(* CODESYS project lclspmps.library
   Company: SLAC
   Version: 0.0.0
   Placeholder: LCLS PMPS
   Title: LCLS PMPS

Project tree, tasks and I/O mapping:
  libraries: LCLS General, * (SLAC); Tc2_MC2, * (Beckhoff Automation GmbH); Tc2_Standard, * (Beckhoff Automation GmbH); Tc2_System, * (Beckhoff Automation GmbH); Tc2_Utilities, * (Beckhoff Automation GmbH); Tc3_Module, * (Beckhoff Automation GmbH); TcUnit, * (www.tcunit.org); VisuDialogs, * (System); VisuSymbols, 3.5.10.0 (System)
  DUTs/
    data type E_ExampleDeviceStates
    data type ST_BeamParams
    data type ST_BinarySolidAttenuator
    data type ST_Device
    data type ST_DeviceState
    data type ST_DeviceStateExt
    data type ST_SolidAttenuatorBlade
  GVLs/
    global variables GVL
    global variables PMPS_GVL_BeamParams
  POUs/
    DeviceImplementationEx1/
      function block FB_ExampleDevice [FBD]: Initialize
      function block FB_ExampleDeviceSM [UML]: AwaitingBeamParameters_ENTRY, ExecutingMove_DO, Moving_ENTRY, Moving_EXIT, NewMove_ENTRY, Stopping_ENTRY, Stopping_EXIT
    DeviceImplementationEx2/
      function block FB_ExampleDeviceSM_All [UML]: Always_DO, AwaitingBeamParameters_ENTRY, Init, MoveComplete_ENTRY, Moving_ENTRY, Moving_EXIT, NewMove_ENTRY, Stopping_ENTRY, Stopping_EXIT, VerifyingNewTargetState_DO
    FlatMirrorEx/
    HelperFunctions/
      function F_DeviceState_To_DeviceStateExt [ST]
      function F_DifferentBeamParams [ST]
      function F_eVWithinSpec [ST]
      function F_SafeBPCompare [ST]
      function F_SetBeamParams [ST]
      function F_SetStateParams [ST]
    MajorComponents/
      function block BeamParameterTransitionManager [UML]: AcquiringSafeBeamParams_DO, AssertFinalBP, AssertTransitionBP, AuthorizeTransition, DeauthorizeMove, DeauthorizeTransition, RemoveTransitionAssertion, RemoveTransitionAuthorization, SetNewTarget, WaitingForFinalAssertion_DO, WaitingForFinalAssertion_EXIT, WaitingForTransitionAssertion_DO, WaitingForTransitionAssertion_EXIT
      function block FB_Arbiter [ST]: A_Init, AddRequest, ArbitrateBP, CheckRequest, GetArbitratedBP, RemoveRequest
      function block FB_BeamClassOutputs [ST]
      function block FB_BeamParamAssertionPool [ST]: A_Add, A_Count, A_GetFirst, A_GetNext, A_Lookup, A_Remove, A_Reset
      function block FB_FastFault [ST]
      function block FB_HardwareFFOutput [ST]: CheckIn, EvaluateOutput, Register
      function block FB_LinearDeviceStateTable [ST]: A_Add, A_Count, A_GetFirst, A_GetNext, A_Lookup, A_Remove, A_Reset
      function block FB_LinearGovernor [ST]
      function block FB_PhotonEnergyWatcher [ST]
      function block FB_UsualSuspects [ST]: M_Register
    TestComponents/
      function block FB_Arbiter_Test [ST]: Arbitration, FB_init, RequestCheckRemoveBP, RunTests
      function block FB_AttenuatorSimulator [ST]
      function block FB_BPTM_Test [ST]: BPTMBasicFunction, FB_init, RunTests
      function block FB_eVWithinSpec_Test [ST]: evWithinRangeChecks, FB_init, RunTests
      function block FB_FastFault_Test [ST]: FB_init, FFCombinedFunctionality, FFRegistration, RunTests
      function block FB_MachineSimulator [ST]
      function block FB_PhotonEnergyWatcher_Test [ST]: FB_init, PEWatcherBasicFunction, RunTests
      function block FB_SafeBPCompare_Test [ST]: BeamOffIsSafe, BPComparisonCheck, FB_init, RunTests
      function block FB_SolidAttenuator [ST]
    program Fast_Faults [ST]
    program Fast_Faults_Evaluate [ST]
    program MachineSimulation [ST]
    program MAIN [ST]: Initialize
    program PMPS_Arbiter [ST]
    program TestSetups [ST]
  VISUs/
    visualisation ArbiterStats
    visualisation FastFaultGUI
    visualisation ImagerGUI
    visualisation PhotonEnergyWatcher
    visualisation Visualization
  text list GlobalTextList
  image pool ImagePool
  00000000-0000-0000-0000-000000000000|MPS Architecture.png
*)

// DUTs/E_ExampleDeviceStates
{attribute 'qualified_only'}
{attribute 'strict'}
TYPE E_ExampleDeviceStates :
(
	enum_member := 0
);
END_TYPE

// DUTs/ST_BeamParams
TYPE ST_BeamParams :
STRUCT
	// Beam parameters
	// These must be filled in by the caller.
	
	//Note: fAtt is a local parameter, meaning it is distributed to the nearest
	// upstream attenuator component.
	fAtt : REAL := 100; //Requested attenuation %
	
	
	
	//Machine parameters
	nBeamClass	:	BYTE := 16#F;
	nRate	:	UDINT	:= 10; //Pulse-rate
	fPP_mJ : REAL := 20; //Per pulse max energy (mJ)
	//1.5-0keV subdivided per bit
	(*
	0.0-0.2 - 0 (lsb)
	0.2-0.3 - 1
	0.3-0.4 - 2
	0.4-0.5 - 3
	0.5-0.6 - 4
	0.6-0.7 - 5
	0.7-0.8 - 6
	0.8-0.9 - 7
	0.9-1.0 - 8
	1.0-1.1 - 9
	1.1-1.2 - 10
	1.2-1.3 - 11
	1.3-1.4 - 12
	1.4-1.5 - 13 (msb)
	na - 14
	na - 15
	*)
	
	{attribute 'displaymode':='binary'}
	neVReqRange	:	WORD	:= 2#1111_1111_1111_1111; //Valid photon energy ranges
	
	reV	:	REAL	:=0; //Photon energy (calculated by undulator gap)

END_STRUCT
END_TYPE

// DUTs/ST_BinarySolidAttenuator
TYPE ST_BinarySolidAttenuator :
STRUCT
	axBlades	: ARRAY [0..9] OF ST_SolidAttenuatorBlade;
END_STRUCT
END_TYPE

// DUTs/ST_Device
TYPE ST_Device :
STRUCT
	//IO
	stAxis	:	AXIS_REF;
	//The following limit switches must be TRUE or high (ie. NC) to enable that direction of motion
	//The EPICS display should show an inverted indicator to communicate end of travel reached
	i_xLoLim	AT %I*	:	BOOL; //Wire normally-closed
	i_xHiLim	AT %I*	:	BOOL; //Wire normally-closed
	
	//Acuator Parameters
	lrUpperPositionLimit	:	LREAL := 10000000000; //Use in conjuntion with limit switches or set to a huge number to ignore
	lrLowerPositionLimit	:	LREAL := -10000000000; //Use in conjuntion with limit switches or set to a huge number to ignore
	
	xEnable	:	BOOL := TRUE;
	
	//Supervisory System
	
	//MPS Override
	xOverrideMPSLimits	: BOOL := FALSE; //Set true to move beyond MPS limits. Note this will trip beam off.
	
	//Status and Faults
	xClearFaults	:	BOOL;	//Rising edge tries to clear faults of all kinds
	
	xGovernorFault	:	BOOL;	//Indicates governor is faulted
	xGovernorOverridden	:	BOOL; //Indicates governor is in override mode
	xSMFault		:	BOOL;	//Indicates component state machine is faulted
	
	//Device States
	StateTable		:	FB_LinearDeviceStateTable;
	
	stTransitionState	:	ST_DeviceState; //The transition state might have non-zero beam parameters
	nSafeState			:	UDINT; //State where the device is considered safe
	nTransitionState	:	UDINT;
	
	nRequestedState	:	UDINT; //EPICS control, cleaned (checked against array limits) and deposited in nTargetState
	nTargetState	:	UDINT; //The requested state should be deposited here after cleaning
	nActiveState	:	UDINT; //The last successfully reached state
	
	
END_STRUCT
END_TYPE

// DUTs/ST_DeviceState
TYPE ST_DeviceState :
STRUCT
	
	//State name
	sStateName	:	STRING;
	nStateRef	:	UDINT; //Primary key of device state database
	
	//////////////////
	// This stuff may belong in a sub-class or something
	//Position
	rPosition	:	REAL := 0; //Center of the state
	//Tolerance
	rTolerance :	REAL := 0; //+/- amount
	//////////////////
	//Required beam parameters
	stReqBeamParam	:	ST_BeamParams;

END_STRUCT
END_TYPE

// DUTs/ST_DeviceStateExt
//Use when working with states in code
//Extended with a valid boolean to indicate the structure was loaded
//properly
TYPE ST_DeviceStateExt EXTENDS ST_DeviceState :
STRUCT
	xValid	:	BOOL := FALSE;
END_STRUCT
END_TYPE

// DUTs/ST_SolidAttenuatorBlade
TYPE ST_SolidAttenuatorBlade :
STRUCT
	xRequestedIn	:	BOOL;
	xCurrentIn	:	BOOL;
	rThickness	:	REAL;
END_STRUCT
END_TYPE

// GVLs/GVL

VAR_GLOBAL
	g_fbArbiter	:	FB_Arbiter;
	g_FastFaultOutput1	:	FB_HardwareFFOutput;
	g_rTestingVelocity	:	LREAL := VISIBLE_TEST_VELOCITY;
	g_fbFFRegistry	:	FB_UsualSuspects;
END_VAR

VAR_GLOBAL CONSTANT
	EXCLUDED_ASSERTION_ID	:	UDINT	:= 16#FFFFFFFF; //An assertion ID that should always return "not found" in the assertion pool
	VISIBLE_TEST_VELOCITY	:	LREAL	:= 10;
	FAST_TEST_VELOCITY		:	LREAL	:= 100;
	MAX_DEVICE_STATES		:	UDINT	:= 300;
END_VAR

// GVLs/PMPS_GVL_BeamParams
{attribute 'qualified_only'}
VAR_GLOBAL
	stReqFBDBeamParamsSum	:	ST_BeamParams;
	stReqMethBeamParamSum	:	ST_BeamParams;
	stCurrentBeamParameters	:	ST_BeamParams;
END_VAR
VAR_GLOBAL CONSTANT
	cstFullBeam	:	ST_BeamParams := (
		fAtt := 0,
		fPP_mJ := 1E4,
		neVReqRange := 2#1111_1111_1111_1111,
		nRate	:= UDINT#1000000
		
);
	cstSafeBeam	:	ST_BeamParams := (
		fAtt := 100,
		fPP_mJ := 0,
		neVReqRange := 0,
		nRate	:= 0
);
	cnMaxStateArrayLen : INT := 20;
	
	MAX_ASSERIONS	:	UDINT := 100; //Maximum number of assertions permitted in the arbiter
	
	g_cBoundaries	:	INT	:= 15;
	g_areVBoundaries	:	ARRAY [0..g_cBoundaries]	OF	REAL	:= [
	0.2,
	0.3,
	0.4,
	0.5,
	0.6,
	0.7,
	0.8,
	0.9,
	1.0,
	1.1,
	1.2,
	1.3,
	1.4,
	1.5,
	1.6
];
END_VAR

// POUs/DeviceImplementationEx1/FB_ExampleDevice
FUNCTION_BLOCK FB_ExampleDevice
VAR_INPUT
END_VAR
VAR_OUTPUT
END_VAR
VAR
	MC_MoveAbsolute_0: MC_MoveAbsolute;
	fbBCTM: BeamParameterTransitionManager;
	FB_ExampleDeviceSM_0: FB_ExampleDeviceSM;
	stDevice	:	ST_Device;
	MC_Power_0: MC_Power;
	MC_Stop_0	:	MC_Stop;
END_VAR

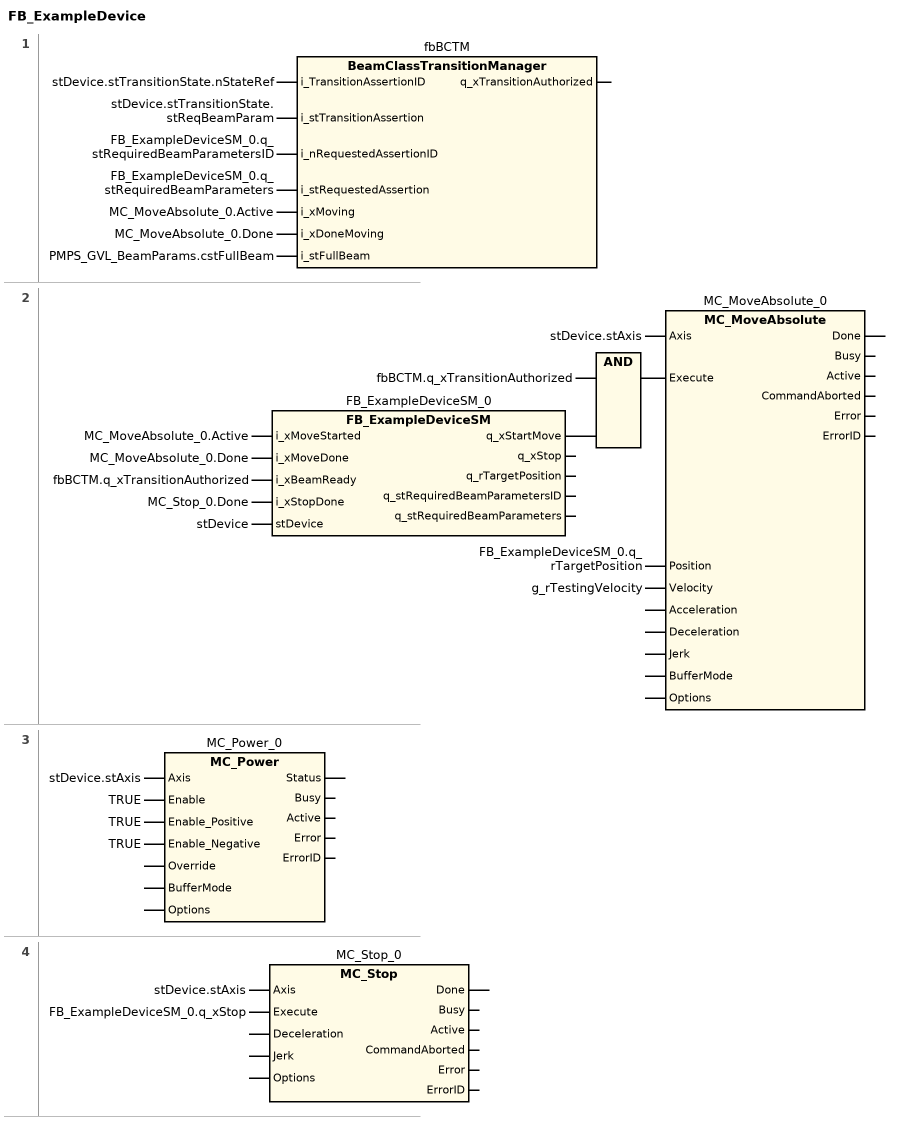
// NETWORK 1
fbBCTM(
    i_TransitionAssertionID := stDevice.stTransitionState.nStateRef,
    i_stTransitionAssertion := stDevice.stTransitionState.stReqBeamParam,
    i_nRequestedAssertionID := FB_ExampleDeviceSM_0.q_stRequiredBeamParametersID,
    i_stRequestedAssertion := FB_ExampleDeviceSM_0.q_stRequiredBeamParameters,
    i_xMoving := MC_MoveAbsolute_0.Active,
    i_xDoneMoving := MC_MoveAbsolute_0.Done,
    i_stFullBeam := PMPS_GVL_BeamParams.cstFullBeam); // BeamClassTransitionManager

// NETWORK 2
FB_ExampleDeviceSM_0(
    i_xMoveStarted := MC_MoveAbsolute_0.Active,
    i_xMoveDone := MC_MoveAbsolute_0.Done,
    i_xBeamReady := fbBCTM.q_xTransitionAuthorized,
    i_xStopDone := MC_Stop_0.Done,
    stDevice := stDevice); // FB_ExampleDeviceSM
MC_MoveAbsolute_0(
    Axis := stDevice.stAxis,
    Execute := fbBCTM.q_xTransitionAuthorized AND FB_ExampleDeviceSM_0.q_xStartMove,
    Position := FB_ExampleDeviceSM_0.q_rTargetPosition,
    Velocity := g_rTestingVelocity); // MC_MoveAbsolute

// NETWORK 3
MC_Power_0(Axis := stDevice.stAxis, Enable := TRUE, Enable_Positive := TRUE, Enable_Negative := TRUE); // MC_Power

// NETWORK 4
MC_Stop_0(Axis := stDevice.stAxis, Execute := FB_ExampleDeviceSM_0.q_xStop); // MC_Stop

ACTION Initialize:

stDevice.astStates[1].rPosition := 100;
stDevice.astStates[1].nStateRef := 16#1;
stDevice.astStates[1].stReqBeamParam := F_SetBeamParams(
	fAtt := 20,
	fPP_mJ := 1,
	fLower_eV := 0,
	fUpper_eV := 1500
);

stDevice.astStates[2].rPosition := 200;
stDevice.astStates[2].nStateRef := 16#2;
stDevice.astStates[2].stReqBeamParam := F_SetBeamParams(
	fAtt := 50,
	fPP_mJ := 1,
	fLower_eV := 0,
	fUpper_eV := 1500
);

stDevice.astStates[3].rPosition := 300;
stDevice.astStates[3].nStateRef := 16#3;
stDevice.astStates[3].stReqBeamParam := F_SetBeamParams(
	fAtt := 50,
	fPP_mJ := 0.5,
	fLower_eV := 0,
	fUpper_eV := 1500
);

stDevice.stTransitionState.nStateRef := 16#10;
stDevice.stTransitionState.stReqBeamParam := F_SetBeamParams(
	fAtt := 100,
	fPP_mJ := 1,
	fLower_eV := 0,
	fUpper_eV := 1500
);
END_ACTION

END_FUNCTION_BLOCK

// POUs/DeviceImplementationEx1/FB_ExampleDeviceSM

FUNCTION_BLOCK FB_ExampleDeviceSM
VAR_INPUT
	i_xMoveStarted	:	BOOL; //Connect to moving flag
	i_xMoveDone	:	BOOL; //Connect to move done flag
	i_xBeamReady	:	BOOL; //Connect to transitioneer
	i_xStopDone	:	BOOL; //Connect to MC_Stop.Done
END_VAR
VAR_OUTPUT
	q_xStartMove	:	BOOL; //Connect to MC_Absolute.Execute
	q_xStop			:	BOOL; //Connect to MC_Stop.Execute
	q_rTargetPosition	:	REAL; //Connect to MC_Absolute.Position
	q_stRequiredBeamParametersID	:	UDINT;
	q_stRequiredBeamParameters	:	ST_BeamParams; //Connect to BeamParameterTransitionManager
END_VAR
VAR_IN_OUT
	stDevice	:	ST_Device;
END_VAR
VAR
	nTargetState	:	INT;
	
	xNewReq	:	BOOL; //Set true when new target request present
	
END_VAR

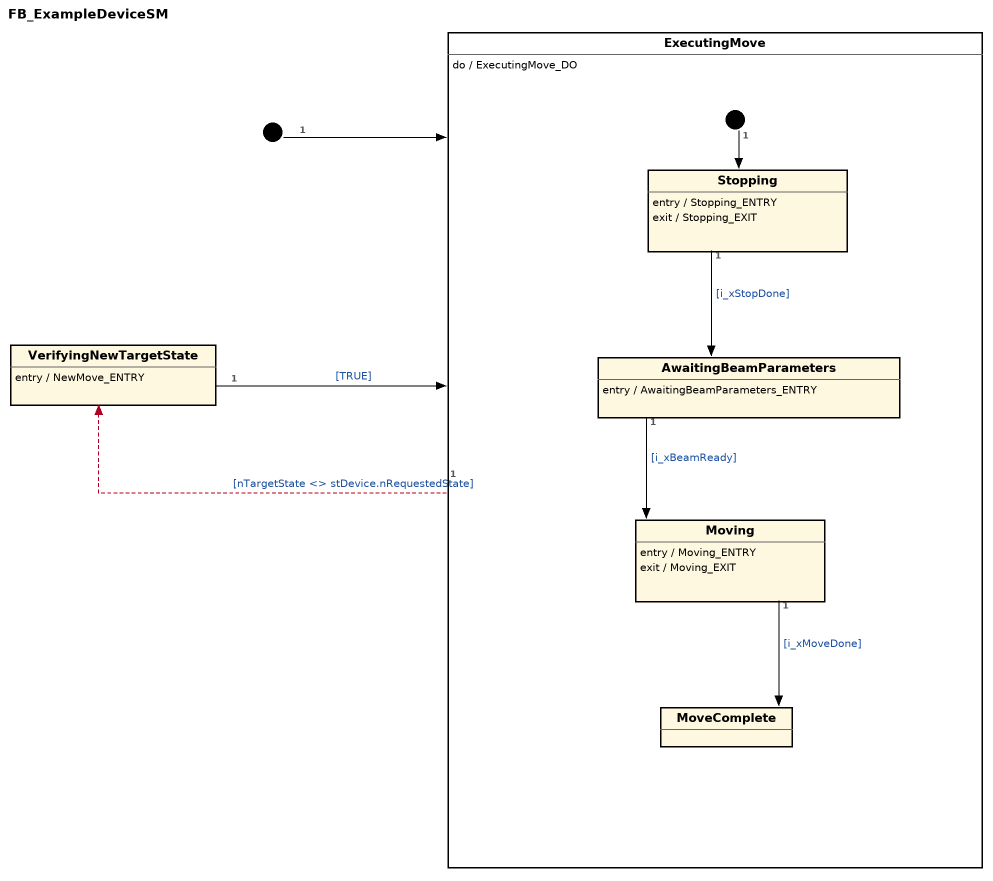
STATECHART FB_ExampleDeviceSM  // abortable
    START StartState1
    COMPOSITE STATE ExecutingMove
        do / ExecutingMove_DO
        START StartState2
        STATE Stopping
            entry / Stopping_ENTRY
            exit / Stopping_EXIT
        STATE AwaitingBeamParameters
            entry / AwaitingBeamParameters_ENTRY
        STATE Moving
            entry / Moving_ENTRY
            exit / Moving_EXIT
        STATE MoveComplete
        StartState2 -> Stopping  // priority 1, on completion
        Stopping -> AwaitingBeamParameters [i_xStopDone] // priority 1, rising edge
        AwaitingBeamParameters -> Moving [i_xBeamReady] // priority 1, rising edge
        Moving -> MoveComplete [i_xMoveDone] // priority 1, rising edge
    END_STATE
    STATE VerifyingNewTargetState
        entry / NewMove_ENTRY
    StartState1 -> ExecutingMove  // priority 1, on completion
    ExecutingMove -> VerifyingNewTargetState [nTargetState <> stDevice.nRequestedState] // priority 1, exception, rising edge
    VerifyingNewTargetState -> ExecutingMove [TRUE] // priority 1
END_STATECHART

ACTION AwaitingBeamParameters_ENTRY:
q_stRequiredBeamParameters := stDevice.astStates[nTargetState].stReqBeamParam;
q_stRequiredBeamParametersID := stDevice.astStates[nTargetState].nStateRef;
END_ACTION

ACTION ExecutingMove_DO:

END_ACTION

ACTION Moving_ENTRY:
q_xStartMove := TRUE;
q_rTargetPosition := stDevice.astStates[nTargetState].rPosition;
END_ACTION

ACTION Moving_EXIT:
q_xStartMove := FALSE;
END_ACTION

ACTION NewMove_ENTRY:

IF stDevice.nRequestedState <= PMPS_GVL_BeamParams.cnMaxStateArrayLen AND
	stDevice.nRequestedState >= 1 THEN
	nTargetState := stDevice.nRequestedState;
END_IF
END_ACTION

ACTION Stopping_ENTRY:
q_xStop	:= TRUE;
END_ACTION

ACTION Stopping_EXIT:
q_xStop := FALSE;
END_ACTION

END_FUNCTION_BLOCK

// POUs/MajorComponents/BeamParameterTransitionManager
(*
Implements the procedure for safely transitioning between device states by asserting the correct beam parameters for 
the state *)
FUNCTION_BLOCK BeamParameterTransitionManager
VAR_IN_OUT
	
	fbArbiter	:	FB_Arbiter; //Connect to local arbiter
	
END_VAR
VAR_INPUT
	i_TransitionAssertionID	:	UDINT := 0;
	i_stTransitionAssertion : ST_BeamParams := PMPS_GVL_BeamParams.cstSafeBeam; //Assertion required during transition (always safer than anything inbetween)
	
	i_nRequestedAssertionID	:	UDINT := 0;
	i_stRequestedAssertion	:	ST_BeamParams := PMPS_GVL_BeamParams.cstSafeBeam; //Requested assertion, change whenever
	
	i_xMoving	:	BOOL := FALSE; //Provide rising edge when device begins moving
	i_xDoneMoving	:	BOOL := FALSE; //Provide rising edge when device is done with a move
	
	stCurrentBeamParameters	:	ST_BeamParams := PMPS_GVL_BeamParams.cstFullBeam; //Connect to current beam parameters
	
END_VAR
VAR_OUTPUT

	q_xTransitionAuthorized	:	BOOL := FALSE; //Rising edge indicating the device is safe to move, use as input to move execute (which requires a rising edge)

END_VAR

VAR
	nTargetAssertionID	:	UDINT := 0;
	stTargetAssertion	:	ST_BeamParams; //Current target assertion
	nCurrentAssertionID	:	UDINT := 0;
	
	xNewBP	:	BOOL;
	xTranBP	:	BOOL;
	xFinalBP	:	BOOL;
	
END_VAR

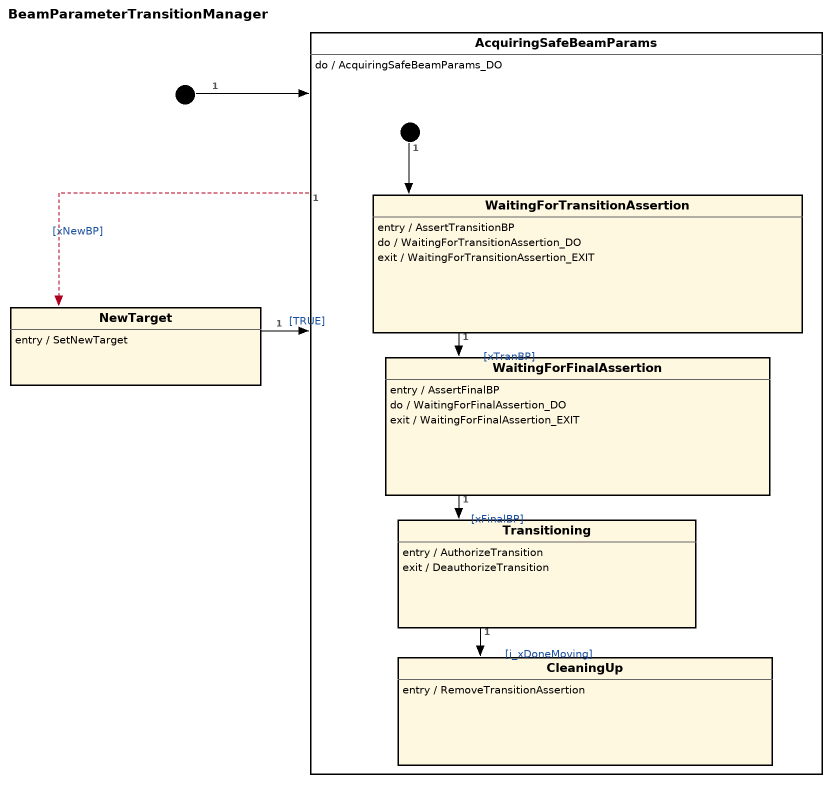
STATECHART BeamParameterTransitionManager  // abortable
    START StartState1_copy
    COMPOSITE STATE AcquiringSafeBeamParams
        do / AcquiringSafeBeamParams_DO
        START StartState1
        STATE WaitingForTransitionAssertion
            entry / AssertTransitionBP
            do / WaitingForTransitionAssertion_DO
            exit / WaitingForTransitionAssertion_EXIT
        STATE WaitingForFinalAssertion
            entry / AssertFinalBP
            do / WaitingForFinalAssertion_DO
            exit / WaitingForFinalAssertion_EXIT
        STATE Transitioning
            entry / AuthorizeTransition
            exit / DeauthorizeTransition
        STATE CleaningUp
            entry / RemoveTransitionAssertion
        StartState1 -> WaitingForTransitionAssertion  // priority 1, on completion
        WaitingForTransitionAssertion -> WaitingForFinalAssertion [xTranBP] // priority 1, rising edge
        WaitingForFinalAssertion -> Transitioning [xFinalBP] // priority 1, rising edge
        Transitioning -> CleaningUp [i_xDoneMoving] // priority 1, rising edge
    END_STATE
    STATE NewTarget
        entry / SetNewTarget
    StartState1_copy -> AcquiringSafeBeamParams  // priority 1, on completion
    AcquiringSafeBeamParams -> NewTarget [xNewBP] // priority 1, exception, rising edge
    NewTarget -> AcquiringSafeBeamParams [TRUE] // priority 1
END_STATECHART

ACTION AcquiringSafeBeamParams_DO:
xNewBP := nTargetAssertionID <> i_nRequestedAssertionID;
END_ACTION

ACTION AssertFinalBP:
//q_stFinalAssertion := stTargetAssertion;

//Clearing previous target parameters
(* This is considered safe at this step as the transition
state beam parameters should always be safer than the
current or target state beam parameters
*)
fbArbiter.RemoveRequest( nCurrentAssertionID );

//Asserting target parameters
fbArbiter.AddRequest(
	nTargetAssertionID,
	stTargetAssertion
);

//Remembering final assertionID for removal later
nCurrentAssertionID := nTargetAssertionID;
END_ACTION

ACTION AssertTransitionBP:

fbArbiter.AddRequest(
	i_TransitionAssertionID,
	i_stTransitionAssertion
);
END_ACTION

ACTION AuthorizeTransition:
q_xTransitionAuthorized := TRUE;
END_ACTION

ACTION DeauthorizeMove:

END_ACTION

ACTION DeauthorizeTransition:
q_xTransitionAuthorized := FALSE;
END_ACTION

ACTION RemoveTransitionAssertion:
//q_stTransitionAssertion := PMPS_GVL_BeamParams.cstFullBeam;

//Removing transition assertion
fbArbiter.RemoveRequest( i_TransitionAssertionID );



//TODO add something to verify removal
END_ACTION

ACTION RemoveTransitionAuthorization:

END_ACTION

ACTION SetNewTarget:
xNewBP := FALSE;
stTargetAssertion := i_stRequestedAssertion;
nTargetAssertionID := i_nRequestedAssertionID;
END_ACTION

ACTION WaitingForFinalAssertion_DO:
//Final Assertion Verification
fbArbiter.CheckRequest( i_nRequestedAssertionID);
xFinalBP := F_SafeBPCompare(stCurrentBeamParameters, stTargetAssertion) AND
	fbArbiter.q_xStateIDFound;
END_ACTION

ACTION WaitingForFinalAssertion_EXIT:
//Set this bool false so we can get a rising edge on the next try
xFinalBP := FALSE;
END_ACTION

ACTION WaitingForTransitionAssertion_DO:
//Transition Assertion Verification
xTranBP	:= F_SafeBPCompare(stCurrentBeamParameters, i_stTransitionAssertion) AND
	fbArbiter.CheckRequest(i_TransitionAssertionID);
END_ACTION

ACTION WaitingForTransitionAssertion_EXIT:
xTranBP := FALSE;
END_ACTION

END_FUNCTION_BLOCK

// POUs/MajorComponents/FB_Arbiter
(* FB Arbiter

The arbiter primary objectives are:
- Provide a simple interface for devices to request beam parameter sets
- Provide a way for devices to verify their BPS is active in the arbiter
- Provide a way for devices remove their requests from evaluation
- Evaluate all active beam parameter requests registered with the aribiter,
to determine the safest combination of all sets, provide this set as an output.
- Do all of this with minimal overhead

To these ends, the arbiter uses a hash-table, the rows being a state-id as the key, and a corresponding
 beam parameter set to be evaluated against all the other sets (or rows), in the table.
 
The hash table can be thought of as an array on steriods, they are worth reading about, suffice to say
the hash table will tell you when you reach the end of all the entries, and enables us to find entries quickly.

These features efficiently address the addition, removal, and verification of beam parameter sets listed in the above requirements.

An important thing to pay attention to is the A_Arbitrate action. This action implements the evaluation of beam parameter
sets against each other.

*)

FUNCTION_BLOCK FB_Arbiter
VAR_INPUT
	i_nStateID	:	UDINT; //Set to the stateID of the state requesting the beam parameter set
	i_stAssertBeamParams	:	ST_BeamParams; //Set to the beam parameter set of the state required
END_VAR
VAR_OUTPUT
	q_stBeamParams	:	ST_BeamParams; //Updated on each cycle of the arbiter FB with the current arbitrated beam parameter set
	
	q_xStateIDFound	:	BOOL; //Set true if a state-id is found in the assertion pool after calling A_VerifyAssertion
END_VAR
VAR
	
	fbBPAssertionPool	:	FB_BeamParamAssertionPool; //Table of active beam parameter assertions
	
	getPosPtr	: POINTER TO T_HashTableEntry := 0; 
	getBPStruct	:	ST_BeamParams;
	stOutputBP	:	ST_BeamParams; //Safest beam parameters from all in the assertion pool
	
	
END_VAR

ACTION A_Init:
// Clears the entire beam parameter assertion pool (hashtable).

fbBPAssertionPool.A_Reset();
END_ACTION

METHOD AddRequest : BOOL
VAR_INPUT
	nStateID	:	DWORD; //StateID of state requesting beam parameter set
	stReqBP		:	ST_BeamParams; //Requested beam params
END_VAR
IF nStateID <> EXCLUDED_ASSERTION_ID THEN
	THIS^.fbBPAssertionPool.A_Add(
		key := nStateID,
		putValue := stReqBP
	);
END_IF
	
IF NOT THIS^.fbBPAssertionPool.bOk THEN
	; //Overflow <TODO>
END_IF

AddRequest := THIS^.fbBPAssertionPool.bOk;
END_METHOD

METHOD ArbitrateBP : ST_BeamParams
VAR_INPUT
	stBP1	:	ST_BeamParams;
	stBP2	:	ST_BeamParams;
END_VAR
//<TODO>Add something here to register the key that won for each param

//Attenuation
ArbitrateBP.fAtt := MAX(stBP1.fAtt, stBP2.fAtt);

//Pulse energy
ArbitrateBP.fPP_mJ := MIN(stBP1.fPP_mJ, stBP2.fPP_mJ);

//Photon energy ranges
ArbitrateBP.neVReqRange := stBP1.neVReqRange AND stBP2.neVReqRange;

//Rate
ArbitrateBP.nRate := MIN(stBP1.nRate, stBP2.nRate);
END_METHOD

(* Searches state assertion pool for a state-id, and sets q_xStateIDFound true if found.

Use like so:

fbArbiter.A_VerifyAssertion(
i_nStateId := nStateIDAssertionToCheck
);

IF fbArbiter.q_xStateIDFound THEN:
	Do something
ELSE:
	Don't do something

*)
METHOD CheckRequest : BOOL
VAR_INPUT
	nReqID	:	DWORD;
END_VAR
THIS^.fbBPAssertionPool.A_Lookup(key := nReqID);

CheckRequest := THIS^.fbBPAssertionPool.bOk;
END_METHOD

METHOD GetArbitratedBP : ST_BeamParams
VAR_INPUT
END_VAR
VAR
	getPosPtr	: POINTER TO T_HashTableEntry := 0;
	getBPStruct	:	ST_BeamParams;
	
	stOutputBP	:	ST_BeamParams; //Holding struct for arbitration process
END_VAR
//Arbitrate
(*
This step cycles through every hash table entry, comparing
the beam parameters from each assertion to what we're planning
to assert.

The safer of the two parameters is kept so at the end we may
have a mix of beam parameters, the composition being safe for
all asserters.

*)

THIS^.fbBPAssertionPool.A_GetFirst( putPosPtr := 0, getPosPtr=>getPosPtr, getValue=>getBPStruct );
IF THIS^.fbBPAssertionPool.bOk THEN //If the table is empty (not OK), we are left with the default stOutputBP set above.
	
	//The first entry in the hash table is taken as the setting to arbitrate against
	stOutputBP := F_SetBeamParams(
		fAtt := getBPStruct.fAtt,
		fPP_mJ := getBPStruct.fPP_mJ,
		neVReqRange	:= getBPStruct.neVReqRange,
		nRate := getBPStruct.nRate
	);

	REPEAT
		THIS^.fbBPAssertionPool.A_GetNext( putPosPtr := THIS^.fbBPAssertionPool.getPosPtr, getPosPtr=>getPosPtr, getValue=>getBPStruct );
		IF THIS^.fbBPAssertionPool.bOk THEN
			stOutputBP := ArbitrateBP(stOutputBP, getBPStruct);
		END_IF
	UNTIL NOT fbBPAssertionPool.bOk
	END_REPEAT
ELSE
	//Safest parameters to start
	stOutputBP := PMPS_GVL_BeamParams.cstSafeBeam;
END_IF

GetArbitratedBP := stOutputBP;
END_METHOD

(* Searches for a state-id, and removes it from the assertion pool.

Use like so:
fbArbiter.A_RemoveAssertion(
i_nStateId := nStateIDAssertionToRemove
);

*)
METHOD RemoveRequest : BOOL
VAR_INPUT
	nReqId	:	DWORD;
END_VAR
IF nReqId <> EXCLUDED_ASSERTION_ID THEN
	THIS^.fbBPAssertionPool.A_Remove(key := nReqId);
	
	IF THIS^.fbBPAssertionPool.bOk THEN
		;
	ELSE
		;
	END_IF
END_IF

RemoveRequest := THIS^.fbBPAssertionPool.bOk;
END_METHOD

END_FUNCTION_BLOCK

// POUs/MajorComponents/FB_BeamParamAssertionPool
(* This function block implements simple database. Data element values are stored in the hash table.  *)
FUNCTION_BLOCK FB_BeamParamAssertionPool
VAR_INPUT
	key 		: DWORD := 0;(* Entry key: used by A_Lookup, A_Remove method, the key variable is also used by A_Add method *)
	putPosPtr	: POINTER TO T_HashTableEntry := 0;(* Hash table entry position pointer (used by A_Find, A_GetNext, A_GetPrev) *)
	putValue 	: ST_BeamParams;(* Hash table entry value (used by A_AddHead, A_AddTail, A_Find )*)
END_VAR
VAR_OUTPUT
	bOk			: BOOL := FALSE;(* TRUE = Success, FALSE = Failed *)
	getPosPtr	: POINTER TO T_HashTableEntry := 0;(* Returned hash table entry position pointer *)
	getValue 	: ST_BeamParams;(* Returned hash table entry value *)
	nCount		: UDINT := 0;(* Hash table size (number of used entries, used by A_Count) *)
END_VAR
VAR
	dataPool	: ARRAY[0..PMPS_GVL_BeamParams.MAX_ASSERIONS] OF ST_BeamParams;(* Structured data element pool *)
	entries		: ARRAY[0..PMPS_GVL_BeamParams.MAX_ASSERIONS] OF T_HashTableEntry;(* Max. number of hash table entries. The value of table entry = 32 bit integer (pointer to dataPool-array-entry) *)
	fbTable 	: FB_HashTableCtrl;(* basic hash table control function block *)
	hTable 		: T_HHASHTABLE;(* hash table handle *)
	pRefPtr		: POINTER TO ST_BeamParams := 0;
	indexOfElem	: ULINT;(* Integer value (max. size: x86=>32bit, x64=>64bit)*)
END_VAR

;

ACTION A_Add:
(* Adds entry to the table *)
MEMSET( ADR( getValue ), 0, SIZEOF( getValue ) );
getPosPtr := 0;

fbTable.A_Add( hTable := hTable, key := key, putValue := ADR(PMPS_GVL_BeamParams.cstSafeBeam)(* we will set this value later *), getPosPtr=>getPosPtr, bOk=>bOk );(* Add new element to the table, getPosPtr points to the new entry *)
IF fbTable.bOk THEN(* Success *)
	fbTable.A_GetIndexAtPosPtr( hTable := hTable, putPosPtr := getPosPtr, getValue =>indexOfElem, bOk=>bOk );(* Get array index of getPosPtr entry *)
	IF fbTable.bOk THEN(* Success *)
		pRefPtr 	:= ADR( dataPool[indexOfElem] );(* Get pointer to the data element *)

		pRefPtr^ := putValue;(* copy application value *)

		fbTable.A_Add( hTable := hTable, key := key, putValue := pRefPtr, bOk=>bOk );(* Assign the entry value = pointer to the data element *)
		IF fbTable.bOk THEN(* Success *)
			getValue := putValue;
		END_IF
	END_IF
END_IF
END_ACTION

ACTION A_Count:
(* Count number of used entries *)
nCount := hTable.nCount;
bOk := TRUE;
END_ACTION

ACTION A_GetFirst:
(* Get first entry position pointer and value *)
MEMSET( ADR( getValue ), 0, SIZEOF( getValue ) );
getPosPtr := 0;

fbTable.A_GetFirst( hTable := hTable, putPosPtr := putPosPtr, getValue=>pRefPtr, getPosPtr=>getPosPtr, bOk=>bOk );
IF fbTable.bOk THEN
	getValue := pRefPtr^;
END_IF
END_ACTION

ACTION A_GetNext:
(* Get next entry position pointer and value *)
MEMSET( ADR( getValue ), 0, SIZEOF( getValue ) );
getPosPtr := 0;
bOk := FALSE;

IF putPosPtr = 0 THEN
	RETURN;
END_IF

fbTable.A_GetNext( hTable := hTable, putPosPtr := putPosPtr, getValue=>pRefPtr, getPosPtr=>getPosPtr, bOk=>bOk );
IF fbTable.bOk THEN
	getValue := pRefPtr^;
END_IF
END_ACTION

ACTION A_Lookup:
(* Lookup for entry by key  *)
MEMSET( ADR( getValue ), 0, SIZEOF( getValue ) );
getPosPtr := 0;

fbTable.A_Lookup( key := key, hTable := hTable, putPosPtr := putPosPtr, getValue=>pRefPtr, getPosPtr=>getPosPtr, bOk=>bOk );
IF fbTable.bOk THEN
	getValue := pRefPtr^;
END_IF
END_ACTION

ACTION A_Remove:
(* Search for entry and remove it *)
MEMSET( ADR( getValue ), 0, SIZEOF( getValue ) );
getPosPtr := 0;

fbTable.A_Remove( key := key, hTable := hTable, putPosPtr := putPosPtr, getValue=>pRefPtr, getPosPtr=>getPosPtr, bOk=>bOk );
IF fbTable.bOk THEN
	getValue := pRefPtr^;
END_IF
END_ACTION

ACTION A_Reset:
(* Reset/initialize linked list *)
MEMSET( ADR( getValue ), 0, SIZEOF( getValue ) );
getPosPtr := 0;
bOk := F_CreateHashTableHnd( ADR( entries ), SIZEOF( entries ), hTable );(* Intialize table handle *)
fbTable.A_Reset( hTable := hTable, bOk=>bOk );
nCount := 0;
END_ACTION

END_FUNCTION_BLOCK

// POUs/HelperFunctions/F_SetBeamParams
FUNCTION F_SetBeamParams : ST_BeamParams
VAR_INPUT
	fAtt	:	REAL := 100;
	fPP_mJ: REAL := 0;
	neVReqRange	:	WORD := 0;
	nRate	:	UDINT := 0;
END_VAR
VAR
	BeamParams	:	ST_BeamParams;
	
END_VAR

BeamParams.fAtt := LIMIT(0,fAtt,100);
BeamParams.fPP_mJ := LIMIT(0,fPP_mJ,20);
BeamParams.neVReqRange := neVReqRange;
BeamParams.nRate	:= MIN(nRate,1000000);

F_SetBeamParams	:= BeamParams;

END_FUNCTION

// POUs/HelperFunctions/F_SafeBPCompare
(*Compares BeamParam1 to BeamParam2: if the parameters of BeamParam1 are more conservative than BeamParam2
the result will be true. *)
FUNCTION F_SafeBPCompare : BOOL
VAR_INPUT
	BeamParam1	:	ST_BeamParams; //Must be more conservative than 2
	BeamParam2	:	ST_BeamParams;
END_VAR
VAR
	// Internal Attenuation OK boolean
	xAttOK: BOOL := FALSE;
	// Internal Per-pulse energy OK boolean
	xPPmjOK: BOOL := FALSE;
	// Internal photon energy OK boolean
	xEvOK: BOOL := FALSE;
	// Internal Beam Rate OK boolean
	xRateOK: BOOL;
	// Beam-rate is zero, masks all others considerations.
	xZeroRate: BOOL;
END_VAR

xAttOK := BeamParam1.fAtt >= BeamParam2.fAtt;
xPPmjOK := BeamParam1.fPP_mJ <= BeamParam2.fPP_mJ;
xEvOK := F_eVWithinSpec(BeamParam1.reV, BeamParam2.neVReqRange);
xZeroRate	:= BeamParam1.nRate = 0;
xRateOK	:= BeamParam1.nRate <= BeamParam2.nRate;

F_SafeBPCompare := xZeroRate OR (xAttOK AND xPPmjOK AND xEvOK AND xRateOK);

END_FUNCTION

// POUs/HelperFunctions/F_eVWithinSpec
//reV must be within permitted range.
FUNCTION F_eVWithinSpec : BOOL
VAR_INPUT
	reV	:	REAL;	//Photon energy to check if within permitted range
	nPermittedRange	:	WORD; //Permitted range
END_VAR
VAR
	//Holding register for permitted ranges
	nPermittedRangeHolding	:	WORD; 
	//For loop counter
	nIndex	:	INT;
	// Lower boundary for range check
	rPreviousBoundary: REAL := 0;
END_VAR

(* How this works:
The within range bool is initialized to false.
Load the word representation of ranges into a holding register.
If the bit at position zero of the holding register is true, and the input eV is
below the boundary at the index position of the boundary array, and the previous boundary
(which initializes at 0), then the within range bool is set. 
Then, we stash the upper boundary as the lower boundary for the next comparison,
and shift the holding register right, which moves the next bit to the zero position.
*)
nPermittedRangeHolding := nPermittedRange;

FOR nIndex := 0 TO PMPS_GVL_BeamParams.g_cBoundaries DO
		
	F_eVWithinSpec S= nPermittedRangeHolding.0 AND( 
		(reV <= PMPS_GVL_BeamParams.g_areVBoundaries[nIndex]*1000) AND
		(reV >= rPreviousBoundary*1000) );
		
	IF F_eVWithinSpec THEN RETURN; END_IF
	
	rPreviousBoundary := PMPS_GVL_BeamParams.g_areVBoundaries[nIndex];
	nPermittedRangeHolding := SHR(nPermittedRangeHolding, 1);
END_FOR

END_FUNCTION

// POUs/DeviceImplementationEx2/FB_ExampleDeviceSM_All
(* This version of the block is self contained. Minimizes wiring.*)
FUNCTION_BLOCK FB_ExampleDeviceSM_All
VAR_INPUT
	cBase: UDINT;
END_VAR
VAR_OUTPUT
END_VAR
VAR_IN_OUT
	fbFastFaultOutput	:	FB_HardwareFFOutput;
	fbArbiter	:	FB_Arbiter;
END_VAR
VAR
	stDevice	:	ST_Device;
	fbGovernor	:	FB_LinearGovernor;
	mcPower	:	MC_Power;
	mcStop: MC_Stop;
	mcAbsolute	:	MC_MoveAbsolute;
	fbBPTM	:	BeamParameterTransitionManager;
	xStartMove: BOOL;
	
	stCheckState: ST_DeviceState;
	stTargetState	:	ST_DeviceState; //Target device state

END_VAR
VAR PERSISTENT
	nLastActiveState	:	UDINT;
END_VAR

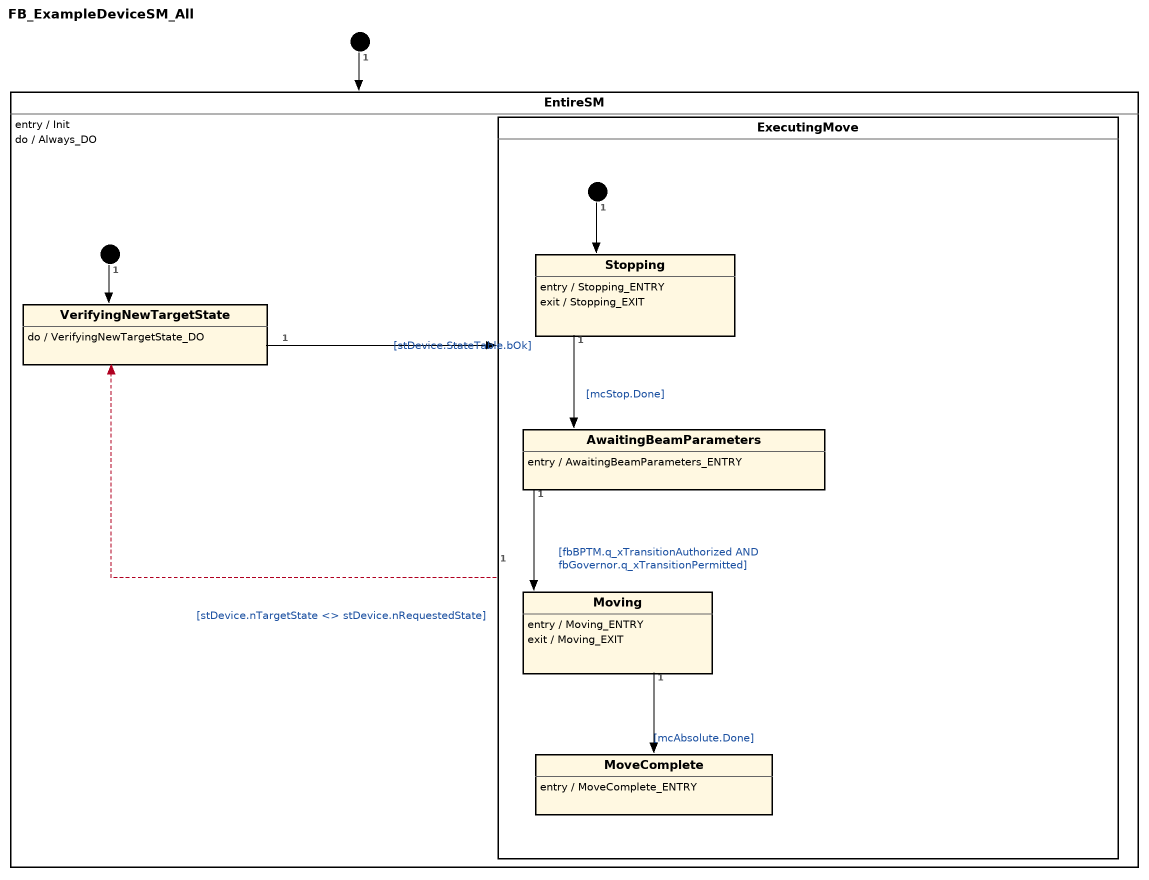
STATECHART FB_ExampleDeviceSM_All  // abortable
    START StartState3
    COMPOSITE STATE EntireSM
        entry / Init
        do / Always_DO
        START StartState1
        COMPOSITE STATE ExecutingMove
            START StartState2
            STATE Stopping
                entry / Stopping_ENTRY
                exit / Stopping_EXIT
            STATE AwaitingBeamParameters
                entry / AwaitingBeamParameters_ENTRY
            STATE Moving
                entry / Moving_ENTRY
                exit / Moving_EXIT
            STATE MoveComplete
                entry / MoveComplete_ENTRY
            StartState2 -> Stopping  // priority 1, on completion
            Stopping -> AwaitingBeamParameters [mcStop.Done] // priority 1, rising edge
            AwaitingBeamParameters -> Moving [fbBPTM.q_xTransitionAuthorized AND fbGovernor.q_xTransitionPermitted] // priority 1, rising edge
            Moving -> MoveComplete [mcAbsolute.Done] // priority 1, rising edge
        END_STATE
        STATE VerifyingNewTargetState
            do / VerifyingNewTargetState_DO
        StartState1 -> VerifyingNewTargetState  // priority 1, on completion
        ExecutingMove -> VerifyingNewTargetState [stDevice.nTargetState <> stDevice.nRequestedState] // priority 1, exception, rising edge
        VerifyingNewTargetState -> ExecutingMove [stDevice.StateTable.bOk] // priority 1
    END_STATE
    StartState3 -> EntireSM  // priority 1, on completion
END_STATECHART

ACTION Always_DO:
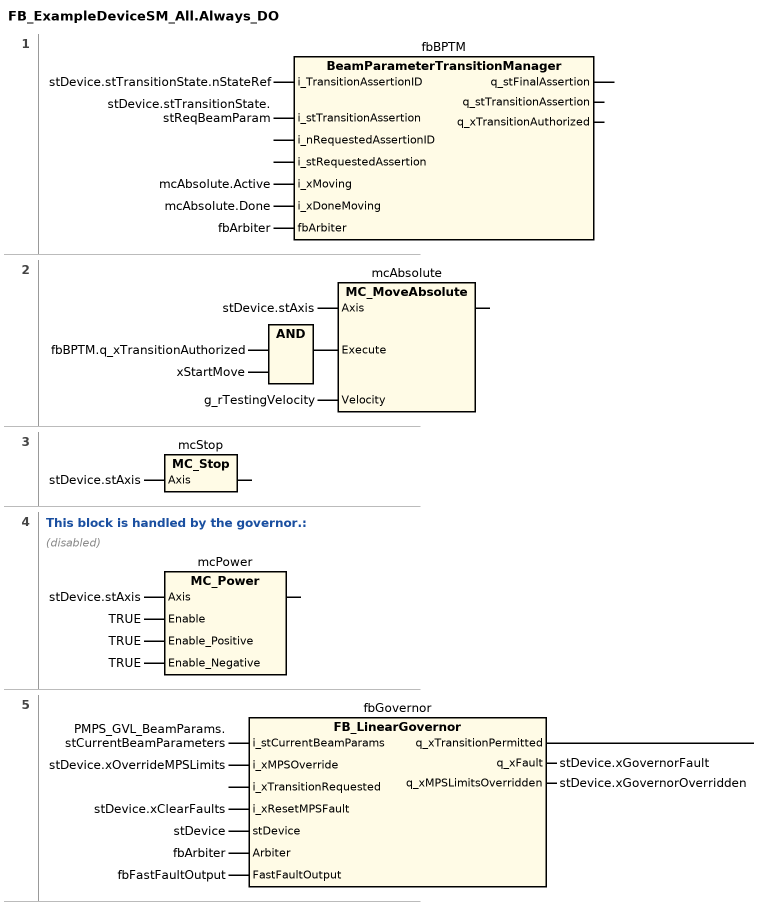
// NETWORK 1
fbBPTM(
    i_TransitionAssertionID := stDevice.stTransitionState.nStateRef,
    i_stTransitionAssertion := stDevice.stTransitionState.stReqBeamParam,
    i_xMoving := mcAbsolute.Active,
    i_xDoneMoving := mcAbsolute.Done,
    fbArbiter := fbArbiter); // BeamParameterTransitionManager

// NETWORK 2
mcAbsolute(
    Axis := stDevice.stAxis,
    Execute := fbBPTM.q_xTransitionAuthorized AND xStartMove,
    Velocity := g_rTestingVelocity); // MC_MoveAbsolute

// NETWORK 3
mcStop(Axis := stDevice.stAxis); // MC_Stop

// NETWORK 4 (disabled)
// label: This block is handled by the governor.
// mcPower(Axis := stDevice.stAxis, Enable := TRUE, Enable_Positive := TRUE, Enable_Negative := TRUE); // MC_Power

// NETWORK 5
fbGovernor(
    i_stCurrentBeamParams := PMPS_GVL_BeamParams.stCurrentBeamParameters,
    i_xMPSOverride := stDevice.xOverrideMPSLimits,
    i_xResetMPSFault := stDevice.xClearFaults,
    stDevice := stDevice,
    Arbiter := fbArbiter,
    FastFaultOutput := fbFastFaultOutput,
    q_xFault => stDevice.xGovernorFault,
    q_xMPSLimitsOverridden => stDevice.xGovernorOverridden); // FB_LinearGovernor
END_ACTION

ACTION AwaitingBeamParameters_ENTRY:
fbBPTM.i_stRequestedAssertion := stTargetState.stReqBeamParam;
fbBPTM.i_nRequestedAssertionID := stTargetState.nStateRef;

//Tell the governor that we're trying to move.
fbGovernor.i_xTransitionRequested := TRUE;
END_ACTION

ACTION Init:

//Safe State
stDevice.nSafeState := cBase;
stDevice.nTransitionState := cBase+100;

//Initialize the State Table
stDevice.StateTable.A_Reset();

//Device State Table Instantiation
//To be done by the device state table database system
F_SetStateParams(
	nStateRef := stDevice.nSafeState,
	rPosition := 0,
	rTolerance := 10,
	stBeamParams := PMPS_GVL_BeamParams.cstFullBeam,
	Table := stDevice.StateTable
);
F_SetStateParams(
	nStateRef := cBase + 1,
	rPosition := 100,
	rTolerance := 10,
	stBeamParams := F_SetBeamParams(
		fAtt := 20,
		fPP_mJ := 1,
		neVReqRange	:= 2#1111_1011_1111_0000,
		nRate := 10
		),
	Table := stDevice.StateTable
);
F_SetStateParams(
	nStateRef := cBase + 2,
	rPosition := 200,
	rTolerance := 10,
	stBeamParams := F_SetBeamParams(
		fAtt := 30,
		fPP_mJ := 1,
		neVReqRange	:= 2#1111_1011_1111_0000,
		nRate := 10
		),
	Table := stDevice.StateTable
);
F_SetStateParams(
	nStateRef := cBase + 3,
	rPosition := 300,
	rTolerance := 10,
	stBeamParams := F_SetBeamParams(
		fAtt := 20,
		fPP_mJ := 1,
		neVReqRange	:= 2#1111_1011_1111_0000,
		nRate := 10
		),
	Table := stDevice.StateTable
);

F_SetStateParams(
	nStateRef := stDevice.nTransitionState,
	rPosition := 0,
	rTolerance := 0,
	stBeamParams := F_SetBeamParams(
		fAtt := 0,
		fPP_mJ := 0,
		neVReqRange	:= 2#1111_1011_1111_0000,
		nRate := 0
		),
	Table := stDevice.StateTable
);

//Set device transition state
stDevice.StateTable.A_Lookup(
	key := stDevice.nTransitionState,
	getValue => stDevice.stTransitionState
);

//Need an initialization routine for setting the active state
//Check if the device is at safe state
//If the device is within the state boundaries, it's considered to be in that state
stDevice.StateTable.A_Lookup(key:= stDevice.nSafeState);
IF stDevice.StateTable.bOk THEN
	stCheckState := stDevice.StateTable.getValue;
ELSE
	stCheckState := stDevice.stTransitionState; //This needs to be safer <TODO>
END_IF

IF stDevice.stAxis.NcToPlc.ActPos <= stCheckstate.rPosition + stCheckState.rTolerance AND
	stDevice.stAxis.NcToPlc.ActPos >= stCheckState.rPosition - stCheckState.rTolerance THEN
	stDevice.nActiveState := nLastActiveState;
ELSE
	stDevice.nActiveState := stDevice.nTransitionState;
END_IF

//Simulation Hardware Limit Switches
stDevice.i_xHiLim := TRUE;
stDevice.i_xLoLim := TRUE;
END_ACTION

ACTION MoveComplete_ENTRY:
//Clear transition request
fbGovernor.i_xTransitionRequested := FALSE;
//Latch active state
stDevice.nActiveState := stDevice.nTargetState;
nLastActiveState := stDevice.nActiveState;
END_ACTION

ACTION Moving_ENTRY:
xStartMove := TRUE;
mcAbsolute.Position := stTargetState.rPosition;
END_ACTION

ACTION Moving_EXIT:
xStartMove := FALSE;
END_ACTION

ACTION NewMove_ENTRY:

END_ACTION

ACTION Stopping_ENTRY:
mcStop.Execute := TRUE;
END_ACTION

ACTION Stopping_EXIT:
mcStop.Execute := FALSE;
END_ACTION

ACTION VerifyingNewTargetState_DO:
stDevice.StateTable.A_Lookup(
	key := stDevice.nRequestedState
);

IF stDevice.StateTable.bOk THEN
	stTargetState := stDevice.StateTable.getValue;
	stDevice.nTargetState := stDevice.nRequestedState;
ELSE
	; //log ignored state/ generate an error? <TODO>
END_IF
END_ACTION

END_FUNCTION_BLOCK

// POUs/MajorComponents/FB_HardwareFFOutput

FUNCTION_BLOCK FB_HardwareFFOutput
VAR_INPUT
	i_xReset	:	BOOL;
	i_xVeto	:	BOOL;	
END_VAR
VAR_OUTPUT
	q_xFastFaultOut	AT %Q*	:	BOOL;
END_VAR
VAR
	xOK	:	BOOL;
	rtReset	:	R_TRIG;
	
	//Fault registration list
	//Fast faults add their name here to indicate they
	//"check in" to indicate their status with this fast
	//fault output. ie. They may be a culprit of beam off.
	asList	:	ARRAY[0..cMaxList] OF T_MaxString;
	nIndex	:	INT;
END_VAR
VAR CONSTANT
	cMaxList	:	INT := 99;
END_VAR

rtReset(CLK:=i_xReset);
xOK S= rtReset.Q;

METHOD CheckIn : BOOL
VAR_INPUT
	i_xOK	:	BOOL; //Keep true to keep beam
END_VAR
IF NOT i_xOK THEN
	THIS^.xOK := FALSE; //Very clever, thanks Zach!
END_IF
END_METHOD

ACTION EvaluateOutput:
q_xFastFaultOut := xOK OR i_xVeto;
END_ACTION

METHOD Register : BOOL
VAR_INPUT
	i_sFFName	:	STRING; //Fast fault FB variable name to register
END_VAR

VAR
END_VAR
IF THIS^.nIndex <= THIS^.cMaxList THEN
	THIS^.asList[MIN(THIS^.nIndex,THIS^.cMaxList)]:=i_sFFName;
	THIS^.nIndex := THIS^.nIndex + 1;
	Register := TRUE; //Add successful
ELSE
	Register := FALSE; //failed to add name to list
END_IF
END_METHOD

END_FUNCTION_BLOCK

// POUs/MajorComponents/FB_LinearGovernor

(* The governor is meant to check your work and keep you from making mistakes.

Checks:
Does your state match the device position and visa versa?
Are the beam parameters safe for the device state?
Did you properly assert the transition and final beam parameters?

*)
FUNCTION_BLOCK FB_LinearGovernor
VAR_INPUT
	i_stCurrentBeamParams	:	ST_BeamParams; //Link to global beam params
	i_xMPSOverride			:	BOOL; //True releases MPS limits after a delay
	i_xTransitionRequested	:	BOOL; //Set true to request a transition
	i_xResetMPSFault	:	BOOL; //Set true to clear MPS fault 
END_VAR
VAR_OUTPUT
	 //True when governor has released restrictions
	q_xTransitionPermitted	:	BOOL;
	//Set if MC_Power has an error, or override mode is requested
	q_xFault	:	BOOL; 
	// Indicates override mode is active
	q_xMPSLimitsOverridden: BOOL;
END_VAR
VAR_IN_OUT
	stDevice	:	ST_Device; //The governed
	Arbiter	:	FB_Arbiter;
	FastFaultOutput	:	FB_HardwareFFOutput;
END_VAR
VAR
	mcPower	:	MC_Power;
	
	xActuatorPositiveEnable: BOOL;
	xActuatorNegativeEnable: BOOL;
	
	xMPSPositiveEnable	:	BOOL;
	xMPSNegativeEnable	:	BOOL;
	lrPosition: LREAL;
	
	lrLatchedTargetPosition	:	LREAL;
	lrLatchedTargetTolerance	:	LREAL;
	stLatchedTargetState	:	ST_DeviceStateExt;
	
	lrMPSUpperLimit: LREAL;
	lrMPSLowerLimit: LREAL;
	rtNewState: R_TRIG;
	xTransitionOK: BOOL;
	
	tonMPSOverrideMode	:	TON := (
		PT := T#5S
	);
	
	srMPSFault	:	SR;
	// Actuator out of bounds fault
	xActuatorOOB: BOOL;
	//Beam parameters out of spec
	xBeamParamsOOS: BOOL;
	//Beam parameters of currently latched state
	
	stLatchedBeamParams: ST_BeamParams;
	stTargetState: ST_DeviceStateExt;
	
	rtLatchNewState	:	R_TRIG;
	xInit: BOOL := TRUE;
	
	stInitDeviceState: ST_DeviceStateExt;
	// Indicates an error with initialization
	xInitFault: BOOL;
	// Indicates the state could not be found in the state table. There may be something wrong in the device state machine implementation or state table instantiation.
	xStateLookupError: BOOL;
	// A transition needs to be requested at least once before we start latching any state.
	xTransitionHasBeenRequested: BOOL := FALSE;
	ffBeamParamsOK : FB_FastFault;
	ffActuatorBoundsOK	:	FB_FastFault;
END_VAR


lrPosition := stDevice.stAxis.NcToPlc.ActPos; //Actuator position

stDevice.stAxis.ReadStatus();
//Init
(* The init strategy is:
If the device is restored and it's residing at the safe position,
no PMPS faults. *)
////////////////////////////////
	IF xInit THEN
		xInit := FALSE;
		//Use nSafeSate for initialization. 
		stDevice.StateTable.A_Lookup(key := stDevice.nSafeState);
		IF stDevice.StateTable.bOk THEN
			stInitDeviceState := F_DeviceState_To_DeviceStateExt(stDevice.StateTable.getValue, TRUE);
			xInitFault := FALSE;
		ELSE
			xInitFault := TRUE;
			stInitDeviceState.xValid := FALSE;
		END_IF
		lrLatchedTargetPosition := stInitDeviceState.rPosition;
		lrLatchedTargetTolerance := stInitDeviceState.rTolerance;
		stLatchedBeamParams := stInitDeviceState.stReqBeamParam;
	END_IF

// The governor will permit transitions once it verifies the transition assertion is active
// Note the governor does not verify the target state beam params are asserted, perhaps it should <TODO>
////////////////////////////////
	IF i_xTransitionRequested THEN
		xTransitionHasBeenRequested	:= TRUE;
		
		xTransitionOK := Arbiter.CheckRequest( stDevice.stTransitionState.nStateRef) AND F_SafeBPCompare(i_stCurrentBeamParams, stDevice.stTransitionState.stReqBeamParam);
		
		//Set the target state for evaluation in further logic
		stdevice.StateTable.A_Lookup(key := stDevice.nTargetState);
		IF stDevice.StateTable.bOk THEN
			stTargetState := F_DeviceState_To_DeviceStateExt(stDevice.StateTable.getValue, TRUE);
			xStateLookupError := FALSE;
		ELSE
			xStateLookupError := TRUE;
			stTargetState.xValid := FALSE;
		END_IF
	ELSE
		xTransitionOK := FALSE;
	END_IF

(* Note about TransitionRequested

If TransitionRequested goes false during a transition, an MPS fault may be induced. This occurs
because the Actuator Out of Bounds fault will go back to using the original state limits, which
the axis may have already moved beyond.

To avoid this transient fault, make sure your device state machine is implemented such that the 
transition request to the governor block remains high until the target position is reached.
*)

//Determine if a transition is complete and latch the new state
(* A transition is complete when:

Axis at standstill.
Axis within tolerance.
No transition req.

Once these conditions are met, the MPS limits shall re-engage to restrict the
axis motion to the tolerance around the state position and the MPS fault monitors
shall evaluate based on the newly latched target state.
*)

rtLatchNewState(CLK := stDevice.stAxis.Status.StandStill AND
	lrPosition <= stTargetState.rPosition + stTargetState.rTolerance AND
	lrPosition >= stTargetState.rPosition - stTargetState.rTolerance AND
	NOT i_xTransitionRequested AND xTransitionHasBeenRequested);
	
IF rtLatchNewState.Q THEN
	lrLatchedTargetPosition := stTargetState.rPosition;
	lrLatchedTargetTolerance := stTargetState.rTolerance;
	stLatchedBeamParams := stTargetState.stReqBeamParam;
	stLatchedTargetState := stTargetState;
END_IF

//Let other blocks know the governor won't interfer with transitions
q_xTransitionPermitted := xTransitionOK;

//Adjust limit ranges based on active state and current target
IF xTransitionOK THEN
	//Extend range to include target state
	lrMPSUpperLimit := MAX(lrMPSUpperLimit, stTargetState.rPosition + stTargetState.rTolerance);
	lrMPSLowerLimit := MIN(lrMPSLowerLimit, stTargetState.rPosition - stTargetState.rTolerance);
ELSE
	//Calculate the limit positions for MPS based on current state
	lrMPSUpperLimit := lrLatchedTargetPosition + lrLatchedTargetTolerance;
	lrMPSLowerLimit := lrLatchedTargetPosition - lrLatchedTargetTolerance;
END_IF


//MPS override
(* In override mode, the device will be free to move anywhere within it's travel range *)
//Permit motion after a small delay
tonMPSOverrideMode(IN:=i_xMPSOverride OR stDevice.xOverrideMPSLimits, Q=>q_xMPSLimitsOverridden);

//Virtual limit switch evaluation
xActuatorPositiveEnable	:= stDevice.i_xHiLim AND lrPosition <= stDevice.lrUpperPositionLimit;
xActuatorNegativeEnable	:= stDevice.i_xLoLim AND lrPosition >= stDevice.lrLowerPositionLimit;

//Evaluate MPS limit states
xMPSPositiveEnable := lrPosition <= lrMPSUpperLimit;
xMPSNegativeEnable := lrPosition >= lrMPSLowerLimit;

//Final Limit switch evaluation
mcPower.Enable_Positive := xActuatorPositiveEnable AND (tonMPSOverrideMode.Q OR xMPSPositiveEnable);
mcPower.Enable_Negative := xActuatorNegativeEnable AND (tonMPSOverrideMode.Q OR xMPSNegativeEnable);

mcPower(
	Axis := stDevice.stAxis,
	Enable := stDevice.xEnable //link to device enable <TODO>
);



//MPS Faults
//Fault if the beam is unsafe for current state
ffBeamParamsOK(i_xOK:=F_SafeBPCompare(i_stCurrentBeamParams, stLatchedBeamParams), 
				i_xReset:=i_xResetMPSFault,
				io_fbFFHWO := FastFaultOutput);

//Fault if the position is outside of the permitted range
ffActuatorBoundsOK(i_xOK := (lrPosition <= lrMPSUpperLimit AND lrPosition >= lrMPSLowerLimit), 
					i_xReset:=i_xResetMPSFault,
				io_fbFFHWO := FastFaultOutput);


	
//Collect all other faults
q_xFault := NOT ffBeamParamsOK.o_xFFLine OR
	NOT ffActuatorBoundsOK.o_xFFLine OR
	mcPower.Error	OR
	i_xMPSOverride	OR
	xInitFault;

//Any faults trip the fast fault line for this FB	
FastFaultOutput.CheckIn(NOT q_xFault);

END_FUNCTION_BLOCK

// POUs/HelperFunctions/F_DeviceState_To_DeviceStateExt
FUNCTION F_DeviceState_To_DeviceStateExt : ST_DeviceStateExt
VAR_INPUT
	stDeviceState	:	ST_DeviceState;
	xValid	:	BOOL;
END_VAR
VAR
END_VAR

F_DeviceState_To_DeviceStateExt.nStateRef := stDeviceState.nStateRef;
F_DeviceState_To_DeviceStateExt.rPosition	:=	stDeviceState.rPosition;
F_DeviceState_To_DeviceStateExt.rTolerance	:=	stDeviceState.rTolerance;
F_DeviceState_To_DeviceStateExt.sStateName	:= stDeviceState.sStateName;
F_DeviceState_To_DeviceStateExt.stReqBeamParam	:= stDeviceState.stReqBeamParam;
F_DeviceState_To_DeviceStateExt.xValid := xValid;

END_FUNCTION

// POUs/MajorComponents/FB_FastFault
{attribute 'reflection'}
FUNCTION_BLOCK FB_FastFault
VAR_INPUT
	i_xOK		:	BOOL;
	i_xReset	:	BOOL; //resets when i_xOK is true and this is true
END_VAR
VAR_OUTPUT
	o_xFFLine	:	BOOL; //Connect to HW output or another FF input if you like
END_VAR
VAR_IN_OUT
	io_fbFFHWO		:	FB_HardwareFFOutput;
END_VAR
VAR
	{attribute 'instance-path'}
	{attribute 'noinit'}
	sPath	:	T_MaxString;
	
	xInit	:	BOOL :=TRUE;
	bsFF	:	RS;
	rtReset	:	R_TRIG;
	
END_VAR

IF xInit	THEN
	io_fbFFHWO.Register(i_sFFName:=sPath);
	//<TODO> if registration doesn't succeed, send warning to diagnostic
	xInit := FALSE;
END_IF


rtReset(CLK:=i_xReset);
bsFF(SET := rtReset.Q, RESET1:= NOT i_xOK);
o_xFFLine := bsFF.Q1;
io_fbFFHWO.CheckIn(bsFF.Q1);

END_FUNCTION_BLOCK

// POUs/HelperFunctions/F_SetStateParams
FUNCTION F_SetStateParams : BOOL;
VAR_INPUT
	nStateRef	:	UDINT;
	rPosition	:	REAL;
	rTolerance: REAL;
	stBeamParams	:	ST_BeamParams;
END_VAR
VAR_IN_OUT
	Table	:	FB_LinearDeviceStateTable;
END_VAR
VAR
	stDeviceState	:	ST_DeviceState;
	
END_VAR

stDeviceState.nStateRef := nStateRef;
stDeviceState.rPosition := rPosition;
stDeviceState.rTolerance := rTolerance;
stDeviceState.stReqBeamParam := stBeamParams;

Table.A_Add(
	key := nStateRef,
	putValue := stDeviceState
);

F_SetStateParams := Table.bOk;

END_FUNCTION

// POUs/MajorComponents/FB_LinearDeviceStateTable
(* This function block implements simple database. Data element values are stored in the hash table.  *)
FUNCTION_BLOCK FB_LinearDeviceStateTable
VAR_INPUT
	key 		: DWORD := 0;(* Entry key: used by A_Lookup, A_Remove method, the key variable is also used by A_Add method *)
	putPosPtr	: POINTER TO T_HashTableEntry := 0;(* Hash table entry position pointer (used by A_Find, A_GetNext, A_GetPrev) *)
	putValue 	: ST_DeviceState;(* Hash table entry value (used by A_AddHead, A_AddTail, A_Find )*)
END_VAR
VAR_OUTPUT
	bOk			: BOOL := FALSE;(* TRUE = Success, FALSE = Failed *)
	getPosPtr	: POINTER TO T_HashTableEntry := 0;(* Returned hash table entry position pointer *)
	getValue 	: ST_DeviceState;(* Returned hash table entry value *)
	nCount		: UDINT := 0;(* Hash table size (number of used entries, used by A_Count) *)
END_VAR
VAR
	dataPool	: ARRAY[0..MAX_DEVICE_STATES] OF ST_DeviceState;(* Structured data element pool *)
	entries		: ARRAY[0..MAX_DEVICE_STATES] OF T_HashTableEntry;(* Max. number of hash table entries. The value of table entry = 32 bit integer (pointer to dataPool-array-entry) *)
	fbTable 	: FB_HashTableCtrl;(* basic hash table control function block *)
	hTable 		: T_HHASHTABLE;(* hash table handle *)
	pRefPtr		: POINTER TO ST_DeviceState := 0;
	indexOfElem	: ULINT;(* Integer value (max. size: x86=>32bit, x64=>64bit)*)
END_VAR

;

ACTION A_Add:
(* Adds entry to the table *)
MEMSET( ADR( getValue ), 0, SIZEOF( getValue ) );
getPosPtr := 0;

fbTable.A_Add( hTable := hTable, key := key, putValue := ADR(PMPS_GVL_BeamParams.cstSafeBeam)(* we will set this value later *), getPosPtr=>getPosPtr, bOk=>bOk );(* Add new element to the table, getPosPtr points to the new entry *)
IF fbTable.bOk THEN(* Success *)
	fbTable.A_GetIndexAtPosPtr( hTable := hTable, putPosPtr := getPosPtr, getValue =>indexOfElem, bOk=>bOk );(* Get array index of getPosPtr entry *)
	IF fbTable.bOk THEN(* Success *)
		pRefPtr 	:= ADR( dataPool[indexOfElem] );(* Get pointer to the data element *)

		pRefPtr^ := putValue;(* copy application value *)

		fbTable.A_Add( hTable := hTable, key := key, putValue := pRefPtr, bOk=>bOk );(* Assign the entry value = pointer to the data element *)
		IF fbTable.bOk THEN(* Success *)
			getValue := putValue;
		END_IF
	END_IF
END_IF
END_ACTION

ACTION A_Count:
(* Count number of used entries *)
nCount := hTable.nCount;
bOk := TRUE;
END_ACTION

ACTION A_GetFirst:
(* Get first entry position pointer and value *)
MEMSET( ADR( getValue ), 0, SIZEOF( getValue ) );
getPosPtr := 0;

fbTable.A_GetFirst( hTable := hTable, putPosPtr := putPosPtr, getValue=>pRefPtr, getPosPtr=>getPosPtr, bOk=>bOk );
IF fbTable.bOk THEN
	getValue := pRefPtr^;
END_IF
END_ACTION

ACTION A_GetNext:
(* Get next entry position pointer and value *)
MEMSET( ADR( getValue ), 0, SIZEOF( getValue ) );
getPosPtr := 0;
bOk := FALSE;

IF putPosPtr = 0 THEN
	RETURN;
END_IF

fbTable.A_GetNext( hTable := hTable, putPosPtr := putPosPtr, getValue=>pRefPtr, getPosPtr=>getPosPtr, bOk=>bOk );
IF fbTable.bOk THEN
	getValue := pRefPtr^;
END_IF
END_ACTION

ACTION A_Lookup:
(* Lookup for entry by key  *)
MEMSET( ADR( getValue ), 0, SIZEOF( getValue ) );
getPosPtr := 0;

fbTable.A_Lookup( key := key, hTable := hTable, putPosPtr := putPosPtr, getValue=>pRefPtr, getPosPtr=>getPosPtr, bOk=>bOk );
IF fbTable.bOk THEN
	getValue := pRefPtr^;
END_IF
END_ACTION

ACTION A_Remove:
(* Search for entry and remove it *)
MEMSET( ADR( getValue ), 0, SIZEOF( getValue ) );
getPosPtr := 0;

fbTable.A_Remove( key := key, hTable := hTable, putPosPtr := putPosPtr, getValue=>pRefPtr, getPosPtr=>getPosPtr, bOk=>bOk );
IF fbTable.bOk THEN
	getValue := pRefPtr^;
END_IF
END_ACTION

ACTION A_Reset:
(* Reset/initialize linked list *)
MEMSET( ADR( getValue ), 0, SIZEOF( getValue ) );
getPosPtr := 0;
bOk := F_CreateHashTableHnd( ADR( entries ), SIZEOF( entries ), hTable );(* Intialize table handle *)
fbTable.A_Reset( hTable := hTable, bOk=>bOk );
nCount := 0;
END_ACTION

END_FUNCTION_BLOCK

// POUs/HelperFunctions/F_DifferentBeamParams
(*Compares BeamParam1 to BeamParam2, if any parameters of BeamParam1 are different than BeamParam2
the result will be true *)
FUNCTION F_DifferentBeamParams : BOOL
VAR_INPUT
	BeamParam1	:	ST_BeamParams;
	BeamParam2	:	ST_BeamParams;
END_VAR
VAR
	// Internal Attenuation OK boolean
	xAttOK: BOOL := FALSE;
	// Internal Per-pulse energy OK boolean
	xPPmjOK: BOOL := FALSE;
	// Internal photon energy OK boolean
	xEvOK: BOOL := FALSE;
	xRateOK: BOOL;
END_VAR

xAttOK := BeamParam1.fAtt <> BeamParam2.fAtt;
xPPmjOK := BeamParam1.fPP_mJ <> BeamParam2.fPP_mJ;
xEvOK := BeamParam1.neVReqRange <> BeamParam2.neVReqRange;
xRateOK	 := BeamParam1.nRate <> BeamParam2.nRate;


F_DifferentBeamParams := xAttOK OR xPPmjOK OR xEvOK OR xRateOK;

END_FUNCTION

// POUs/MajorComponents/FB_BeamClassOutputs
(*
Sets the beam class assertion lines for a given beam class.
*)
FUNCTION_BLOCK FB_BeamClassOutputs
VAR_INPUT
	i_ArbiterBP	:	ST_BeamParams;
END_VAR
VAR_OUTPUT
END_VAR
VAR
	wBeamClass	:	BYTE;
	q_BC_ASSERTION_LINES	AT	%Q*	: ARRAY [1..16] OF	BOOL;
	InitCounter: INT;
	counter	:	INT;
END_VAR


//Beam Class
////////////////////////////////////
//0x0 = 0000 0000 0000 0000
//0x1 = 0000 0000 0000 0001
//0xF = 1111 1111 1111 1111

//Initialize BC lines to zero on every pass
FOR InitCounter := 1 TO 16 DO
	q_BC_ASSERTION_LINES[InitCounter] := FALSE;
END_FOR

//Set BC lines according to beam class
//A BC of 0x0 would pass over this loop, setting none of the lines high
// , as FOR loops check the initialized variable at the top to see if it's >
// than the "TO" variable.
FOR wBeamClass:=1 TO i_ArbiterBP.nBeamClass DO
	q_BC_ASSERTION_LINES[wBeamClass] := TRUE;
END_FOR

END_FUNCTION_BLOCK

// POUs/MajorComponents/FB_PhotonEnergyWatcher
(*
A. Wallace 4-22-2019
The photon energy watcher ensures the current and target photon energy is within
the arbirated bounds. Target in this case means, the calculated target photon energy
from the PVs that control the mechatronics of the undulators/ the electron energy.

If there are control PVs that match the monitor PVs, the control PVs are used to 
calculate a "target" photon energy. This is supposed to cover when the undulators/
electron energy is transitioning.

The abritrated bounds come from a simple AND of all the permitted ranges. See
the arbitrate action of the arbiter FB.

Note, this protection logic does not account for beam-off when determining fast-fault
status. If a device is requesting a limited range of eV, this request must be honored,
regardless of current beam-rate.
*)
FUNCTION_BLOCK FB_PhotonEnergyWatcher
VAR_INPUT
	i_stCurrentBeamParams	:	ST_BeamParams; //Link to global beam params
	i_stMachineTargetBeamParams	:	ST_BeamParams; //Link to global machine target beam params
	i_stRequestedBeamParams	:	ST_BeamParams; //Link to arbiter output or beam param. requestor
	// Reset fault
	i_xReset: BOOL;
END_VAR
VAR_OUTPUT
END_VAR
VAR_IN_OUT
	io_fbFFHWO	:	FB_HardwareFFOutput;
END_VAR
VAR
	xPhotonEnergyWithinBounds	:	BOOL;
	fbFF	:	FB_FastFault;
END_VAR

xPhotonEnergyWithinBounds := F_eVWithinSpec(i_stCurrentBeamParams.reV, i_stRequestedBeamParams.neVReqRange) AND
							F_eVWithinSpec(i_stMachineTargetBeamParams.reV, i_stRequestedBeamParams.neVReqRange);

fbFF(i_xOK := xPhotonEnergyWithinBounds,
	i_xReset := i_xReset,
	io_fbFFHWO := io_fbFFHWO);

END_FUNCTION_BLOCK

// POUs/MajorComponents/FB_UsualSuspects
//Used to register fast faults
FUNCTION_BLOCK FB_UsualSuspects
VAR_INPUT
END_VAR
VAR_OUTPUT
END_VAR
VAR
	asList	:	ARRAY[0..cMaxList] OF T_MaxString;
	nIndex	:	INT;
END_VAR
VAR CONSTANT
	cMaxList	:	INT := 99;
END_VAR

METHOD M_Register : BOOL
VAR_INPUT
	i_sFFName	:	STRING; //Fast fault FB variable name to register
END_VAR

VAR
END_VAR
IF THIS^.nIndex <= THIS^.cMaxList THEN
	THIS^.asList[MIN(THIS^.nIndex,THIS^.cMaxList)]:=i_sFFName;
	THIS^.nIndex := THIS^.nIndex + 1;
	M_Register := TRUE; //Add successful
ELSE
	M_Register := FALSE; //failed to add name to list
END_IF
END_METHOD

END_FUNCTION_BLOCK

// POUs/TestComponents/FB_Arbiter_Test
{attribute 'call_after_init'}
FUNCTION_BLOCK FB_Arbiter_Test EXTENDS FB_TestSuite IMPLEMENTS I_RunnableTestSuite
VAR_INPUT
END_VAR
VAR_OUTPUT
END_VAR
VAR
	fbAssert : TcUnit.FB_Assert;
END_VAR

METHOD PRIVATE Arbitration
VAR_INPUT
END_VAR
VAR
	fbArbiter	:	FB_Arbiter;
	
 	nAttReqID	:	UDINT	:= 1;
	stAttReqBP	:	ST_BeamParams := PMPS_GVL_BeamParams.cstFullBeam;
	
	nPPEReqID	:	UDINT	:= 2;
	stPPEReqBP	:	ST_BeamParams := PMPS_GVL_BeamParams.cstFullBeam;
	
	nEVReqID	:	UDINT	:= 3;
	stEVReqBP	:	ST_BeamParams := PMPS_GVL_BeamParams.cstFullBeam;
	
	nRateReqID	:	UDINT	:= 4;
	stRateReqBP	:	ST_BeamParams := PMPS_GVL_BeamParams.cstFullBeam;
	
	stArbitratedBP	:	ST_BeamParams;
	stExpectedBP	:	ST_BeamParams := PMPS_GVL_BeamParams.cstFullBeam;
END_VAR
TEST('Arbitration');

//Initialize arbiter
fbArbiter.A_Init();

stAttReqBP.fAtt := 50;
stPPEReqBP.fPP_mJ := 1;
stEVReqBP.neVReqRange := 2#1111_1100_1111_1111;
stRateReqBP.nRate := 120;

//Load arbiter with beam parameter sets
fbAssert.AssertTrue(fbArbiter.AddRequest(nAttReqID, stAttReqBP),
					'Safest attenuation request failed to load');
					
//Load arbiter with beam parameter sets
fbAssert.AssertTrue(fbArbiter.AddRequest(nPPEReqID, stPPEReqBP),
					'Safest PPE request failed to load');
					
//Load arbiter with beam parameter sets
fbAssert.AssertTrue(fbArbiter.AddRequest(nEVReqID, stEVReqBP),
					'Safest stEVReqBP request failed to load');
					
//Load arbiter with beam parameter sets
fbAssert.AssertTrue(fbArbiter.AddRequest(nRateReqID, stRateReqBP),
					'Safest stEVReqBP request failed to load');

stExpectedBP.fAtt 	:= 	stAttReqBP.fAtt;
stExpectedBP.fPP_mJ	:=  stPPEReqBP.fPP_mJ;
stExpectedBP.neVReqRange := stEVReqBP.neVReqRange;
stExpectedBP.nRate := stRateReqBP.nRate;

stArbitratedBP := fbArbiter.GetArbitratedBP();

fbAssert.AssertFalse(F_DifferentBeamParams(stExpectedBP, stArbitratedBP),
				'Arbitrated BP does not match expected.');
END_METHOD

METHOD FB_init : BOOL
VAR_INPUT
	bInitRetains : BOOL; // if TRUE, the retain variables are initialized (warm start / cold start)
	bInCopyCode : BOOL;  // if TRUE, the instance afterwards gets moved into the copy code (online change)
END_VAR
SUPER^.RegisterTestSuite(THIS^);
END_METHOD

METHOD PRIVATE RequestCheckRemoveBP
VAR_INPUT
END_VAR
VAR
	fbArbiter	:	FB_Arbiter;
	
	nId	:	DWORD := 1;
	stReq	:	ST_BeamParams;
END_VAR
fbArbiter.A_Init();

TEST('RequestBP');
fbAssert.AssertTrue(fbArbiter.AddRequest(nId, stReq),
	'Request failed');
	
TEST('DuplicateID');
fbAssert.AssertFalse(fbArbiter.AddRequest(nId, stReq),
	'Duplicate request accepted, not good.');
	
TEST('CheckBP');
fbAssert.AssertTrue(fbArbiter.CheckRequest(nId),
	'Check failed');
	
TEST('IDDoesNotExist');
fbAssert.AssertFalse(fbArbiter.CheckRequest(nId+1),
	'Check returned true when ID does not exist');
	
TEST('RemoveBP');
fbAssert.AssertTrue(fbArbiter.RemoveRequest(nId),
	'Remove failed');
fbAssert.AssertFalse(fbArbiter.CheckRequest(nId),
	'Remove did not remove request');
END_METHOD

METHOD RunTests : TCUNIT.E_TestSuiteRunState
Arbitration();
RequestCheckRemoveBP();

RunTests := TcUnit.E_TestSuiteRunState.FINISHED;
END_METHOD

END_FUNCTION_BLOCK

// POUs/TestComponents/FB_AttenuatorSimulator
FUNCTION_BLOCK FB_AttenuatorSimulator
VAR_INPUT
	i_rRequestedAttenuation	:	REAL;
END_VAR
VAR_OUTPUT
	q_xFault	:	BOOL;
	q_rCurrentAttenuation	:	REAL;
END_VAR
VAR_IN_OUT
	Arbiter	:	FB_Arbiter; //Higher level arbiter from which upstream attenuation can be requested
END_VAR
VAR
	tonDelay	:	TON := (
		PT := T#3S
		);
	rLower_eVThreshold	:	REAL := 300;
END_VAR

// Really basic delay
tonDelay(IN := i_rRequestedAttenuation <> q_rCurrentAttenuation);

IF tonDelay.Q THEN
	q_rCurrentAttenuation := i_rRequestedAttenuation;
END_IF

END_FUNCTION_BLOCK

// POUs/TestComponents/FB_BPTM_Test
{attribute 'call_after_init'}
FUNCTION_BLOCK FB_BPTM_Test EXTENDS FB_TestSuite IMPLEMENTS I_RunnableTestSuite
VAR_INPUT
END_VAR
VAR_OUTPUT
END_VAR
VAR
	fbAssert : TcUnit.FB_Assert;
END_VAR

METHOD PRIVATE BPTMBasicFunction
VAR_INPUT
END_VAR
VAR
	fbBPTM	:	BeamParameterTransitionManager;
	fbArbiter	:	FB_Arbiter;
	
	//Final and transition assertions
	nTransitionID	:	UDINT := 1;
	stTransitionAssertion	:	ST_BeamParams := PMPS_GVL_BeamParams.cstSafeBeam;
	
 	nReqID	:	UDINT	:= 2;
	stReqAssertion	:	ST_BeamParams := PMPS_GVL_BeamParams.cstSafeBeam;
	
	fbMachine	:	FB_MachineSimulator;
END_VAR
//Initialize arbiter
fbArbiter.A_Init();

//Call BPTM with requested final state and transition state
fbBPTM(
	fbArbiter := fbArbiter,
	i_TransitionAssertionID := nTransitionID,
	i_stTransitionAssertion := stTransitionAssertion,
	
	i_nRequestedAssertionID := nReqID,
	i_stRequestedAssertion := stReqAssertion
);

TEST('BPTMAssertsTransitionBeforeFinal');
	
//Second pass should move into waiting for transition assertion, arbiter should have transition id
fbBPTM(fbArbiter:= fbArbiter);

fbAssert.AssertTrue(
	fbBPTM.UML_SC_BeamParameterTransitionManager.States[fbBPTM.UML_SC_BeamParameterTransitionManager.Names.WaitingForTransitionAssertion].Active,
	'BPTM did not move into Waiting for transition assertion'); 
	

fbAssert.AssertTrue(fbArbiter.CheckRequest(nTransitionID), 'Arbiter did not accept BPTM transition assertion');


TEST('BPTM: Arbiter Only Has Transition');
fbAssert.AssertTrue(fbArbiter.CheckRequest(nTransitionID),
	'Arbiter does not have transition assertion.');
	
TEST('BPTM waits for transition BP');	
fbAssert.AssertFalse(fbArbiter.CheckRequest(nReqID),
	'Arbiter already has final ID before transition conditions are met');
	
fbAssert.AssertFalse(fbBPTM.q_xTransitionAuthorized,
	'Transition should not be authorized until the arbiter has final assertion');

TEST('BPTM Requests Final');
fbBPTM(fbArbiter := fbArbiter,
	stCurrentBeamParameters := stTransitionAssertion);
	
fbAssert.AssertTrue(fbArbiter.CheckRequest(nReqID),
	'Final assertion should be in arbiter');
	
TEST('BPTM Authorizes Transition');
fbAssert.AssertTrue(fbBPTM.q_xTransitionAuthorized,
	'Transition should be authorized at this point');
	
TEST('BPTM Current assertion id is set');
fbAssert.AssertEquals(nReqID, fbBPTM.nCurrentAssertionID,
	'nCurrentAssertionID not set.');
	
TEST('BPTM Transition Deauthorized');
fbBPTM(fbArbiter := fbArbiter,
		i_xDoneMoving := TRUE);
fbAssert.AssertFalse(fbBPTM.q_xTransitionAuthorized,
	'Transition authorization should go away when done moving');
	
TEST('BPTM Transition BP request removed');
fbAssert.AssertFalse(fbArbiter.CheckRequest(nTransitionID),
	'Transition ID still in arbiter');
	
//Basic testing is complete, interruption functionality testing next
//Continuing to use the same BPTM because internal variable nCurrentAssertionID is now non-zero
END_METHOD

METHOD FB_init : BOOL
VAR_INPUT
	bInitRetains : BOOL; // if TRUE, the retain variables are initialized (warm start / cold start)
	bInCopyCode : BOOL;  // if TRUE, the instance afterwards gets moved into the copy code (online change)
END_VAR
SUPER^.RegisterTestSuite(THIS^);
END_METHOD

METHOD RunTests : TCUNIT.E_TestSuiteRunState
BPTMBasicFunction();

RunTests := TcUnit.E_TestSuiteRunState.FINISHED;
END_METHOD

END_FUNCTION_BLOCK

// POUs/TestComponents/FB_MachineSimulator
(* Simulates the machine responding to requests by adding a bit of delay/ ramps
*)
FUNCTION_BLOCK FB_MachineSimulator
VAR_INPUT
	i_stAssertedParams	:	ST_BeamParams;
	i_reV	:	REAL;
	i_xFault	:	BOOL;
END_VAR
VAR_OUTPUT
	q_stMachineParams	:	ST_BeamParams;
END_VAR
VAR
	fTargetAtt: REAL;
	tonAttTimer	:	TON := (
		PT := T#2S
		);
	fTargetPP_mJ: REAL;
	tonPPETimer: TON := (
		PT := T#2S
	);
END_VAR


//Attenuation
IF i_stAssertedParams.fAtt <> fTargetAtt THEN
	tonAttTimer(IN:=FALSE);
	fTargetAtt := i_stAssertedParams.fAtt;
ELSIF NOT tonAttTimer.Q THEN
	tonAttTimer(IN:=TRUE);
ELSE
	q_stMachineParams.fAtt := fTargetAtt;
END_IF

//Pulse Energy
IF i_stAssertedParams.fPP_mJ <> fTargetPP_mJ THEN
	tonPPETimer(IN:=FALSE);
	fTargetPP_mJ := i_stAssertedParams.fPP_mJ;
ELSIF NOT tonAttTimer.Q THEN
	tonPPETimer(IN:=TRUE);
ELSE
	q_stMachineParams.fPP_mJ := fTargetPP_mJ;
END_IF

//Photon Energy is set arbitrarily, beyond our control.
q_stMachineParams.reV := i_reV;

//Rate
IF i_xFault THEN
	q_stMachineParams.nRate := 0;
ELSE
	q_stMachineParams.nRate := i_stAssertedParams.nRate;
END_IF

END_FUNCTION_BLOCK

// POUs/TestComponents/FB_eVWithinSpec_Test
{attribute 'call_after_init'}
FUNCTION_BLOCK FB_eVWithinSpec_Test EXTENDS FB_TestSuite IMPLEMENTS I_RunnableTestSuite
VAR_INPUT
END_VAR
VAR_OUTPUT
END_VAR
VAR
	fbAssert : TcUnit.FB_Assert;
END_VAR

METHOD PRIVATE evWithinRangeChecks
VAR_INPUT
END_VAR
VAR

END_VAR
TEST('evWithinRangeChecks');
	
//Upper limit equal
fbAssert.AssertTrue(
	F_eVWithinSpec(300, 2#0000_0000_0000_0010),
	'Upper limit not inclusive');
//Lower limit equal
fbAssert.AssertTrue(
	F_eVWithinSpec(300, 2#0000_0000_0000_0100),
	'Lower limit not inclusive');
//Out of range
fbAssert.AssertFalse(
	F_eVWithinSpec(300.1, 2#0000_0000_0000_0010),
	'Out of range failed, whatever you did, it broke this really bad.');
//Negative eV
fbAssert.AssertFalse(
	F_eVWithinSpec(-300, 16#FFFF),
	'Working with antimatter? Negative eV should not be acceptable.');
//Upper unallocated range
fbAssert.AssertFalse(
	F_eVWithinSpec(1700, 2#1000_0000_0000_0000),
	'eV range should not evaluate past 1.6keV');
END_METHOD

METHOD FB_init : BOOL
VAR_INPUT
	bInitRetains : BOOL; // if TRUE, the retain variables are initialized (warm start / cold start)
	bInCopyCode : BOOL;  // if TRUE, the instance afterwards gets moved into the copy code (online change)
END_VAR
SUPER^.RegisterTestSuite(THIS^);
END_METHOD

METHOD RunTests : TCUNIT.E_TestSuiteRunState
evWithinRangeChecks();

RunTests := TcUnit.E_TestSuiteRunState.FINISHED;
END_METHOD

END_FUNCTION_BLOCK

// POUs/TestComponents/FB_FastFault_Test
{attribute 'call_after_init'}
FUNCTION_BLOCK FB_FastFault_Test EXTENDS FB_TestSuite IMPLEMENTS I_RunnableTestSuite
VAR_INPUT
END_VAR
VAR_OUTPUT
END_VAR
VAR
	fbAssert : TcUnit.FB_Assert;
END_VAR

METHOD FB_init : BOOL
VAR_INPUT
	bInitRetains : BOOL; // if TRUE, the retain variables are initialized (warm start / cold start)
	bInCopyCode : BOOL;  // if TRUE, the instance afterwards gets moved into the copy code (online change)
END_VAR
SUPER^.RegisterTestSuite(THIS^);
END_METHOD

METHOD PRIVATE FFCombinedFunctionality
VAR_INPUT
END_VAR
VAR
	fbFF	:	FB_FastFault;
	fbFFO	:	FB_HardwareFFOutput;
	
END_VAR
TEST('FFCombinedFunctionality');

//Clear initial faults
fbFFO(i_xReset:=TRUE); //Reset requested at start of cycle

fbFF(io_fbFFHWO := fbFFO, //FF reset somehwere in code
	i_xOK := TRUE,
	i_xReset := TRUE);

fbFFO.EvaluateOutput(); //FFO eval called at end of cycle
	
fbAssert.AssertTrue(fbFFO.q_xFastFaultOut,
	'Fast fault did not clear');


//Induce fault with FF

fbFFO(i_xReset := FALSE); //Reset released at start of cycle

fbFF(io_fbFFHWO := fbFFO, //FF faulted
	i_xOK := FALSE); //Reset is still set true from last call.
	
fbFFO.EvaluateOutput(); //FFO eval called at end of cycle

fbAssert.AssertFalse(fbFFO.q_xFastFaultOut,
	'Fast fault did not trip the beam');
	
	
//FFO remains faulted until local (FF) and FFO receieve fresh reset request, and faults
//are actually cleared

//Attempt to clear FFO fails because FF still faulted
fbFFO(i_xReset := TRUE); //Reset requested

fbFF(io_fbFFHWO := fbFFO, //FF faulted
	i_xOK := FALSE,
	i_xReset := FALSE);
	
fbFFO.EvaluateOutput(); //FFO eval called at end of cycle

fbAssert.AssertFalse(fbFFO.q_xFastFaultOut,
	'Fast fault output cleared while fault remains, very bad');
	
//Attempt to clear FF while fault remains fails
fbFFO(i_xReset := FALSE);
fbFFO(i_xReset := TRUE); //Reset requested

fbFF(io_fbFFHWO := fbFFO, //FF faulted
	i_xOK := FALSE,
	i_xReset := TRUE); //This reset should fail.
	
fbFFO.EvaluateOutput(); //FFO eval called at end of cycle

fbAssert.AssertFalse(fbFFO.q_xFastFaultOut,
	'Fast fault cleared while fault remains, very bad');
END_METHOD

METHOD PRIVATE FFRegistration
VAR_INPUT
END_VAR
VAR
	fbFF	:	FB_FastFault;
	fbFFO	:	FB_HardwareFFOutput;
END_VAR
TEST('FFRegistration');

fbFF(io_fbFFHWO := fbFFO);

fbAssert.AssertEquals_STRING(fbFF.sPath, fbFFO.asList[fbFFO.nIndex-1],
	'FF registration with FFO did not succeed');
END_METHOD

METHOD RunTests : TCUNIT.E_TestSuiteRunState
FFRegistration();
FFCombinedFunctionality();

RunTests := TcUnit.E_TestSuiteRunState.FINISHED;
END_METHOD

END_FUNCTION_BLOCK

// POUs/TestComponents/FB_PhotonEnergyWatcher_Test
{attribute 'call_after_init'}
FUNCTION_BLOCK FB_PhotonEnergyWatcher_Test EXTENDS FB_TestSuite IMPLEMENTS I_RunnableTestSuite
VAR_INPUT
END_VAR
VAR_OUTPUT
END_VAR
VAR
	fbAssert : TcUnit.FB_Assert;
END_VAR

METHOD FB_init : BOOL
VAR_INPUT
	bInitRetains : BOOL; // if TRUE, the retain variables are initialized (warm start / cold start)
	bInCopyCode : BOOL;  // if TRUE, the instance afterwards gets moved into the copy code (online change)
END_VAR
SUPER^.RegisterTestSuite(THIS^);
END_METHOD

METHOD PRIVATE PEWatcherBasicFunction
VAR_INPUT
END_VAR
VAR
	fbPEW	:	FB_PhotonEnergyWatcher;
	fbFFO	:	FB_HardwareFFOutput;
	q_Output	:	BOOL;
	
	stCurBeamParams	:	ST_BeamParams;
	stMachineTargetBeamParams	:	ST_BeamParams;
	stReqBeamParams	:	ST_BeamParams;
END_VAR
TEST('PEWatcherBasicFunction');

//Clear FFO fault to start
fbFFO(i_xReset:=TRUE);

//All eV OK
stCurBeamParams.reV := 800;
	
stMachineTargetBeamParams.reV := 800;

stReqBeamParams.neVReqRange := 2#1111_1111_1111_1111;	

fbFFO(i_xReset:=FALSE); //Reset request released
	
fbPEW(i_stCurrentBeamParams := stCurBeamParams,
	i_stMachineTargetBeamParams := stMachineTargetBeamParams,
	i_stRequestedBeamParams := stReqBeamParams,
	io_fbFFHWO := fbFFO,
	i_xReset := TRUE); //Clear local FF within PEW
	
fbFFO.EvaluateOutput(q_xFastFaultOut=>q_Output); //This simulates a completed PLC cycle
//Evaluate output should be called once at the end of a PLC cycle.

fbAssert.AssertTrue(q_Output,
	'Beam within limits, FFO should be true');
	
	
//Req eV moved out of range
stCurBeamParams.reV := 800;
	
stMachineTargetBeamParams.reV := 800;

stReqBeamParams.neVReqRange := 2#0000_1111_0011_1111;

fbPEW.i_xReset := FALSE; //release local FF reset req	
fbPEW(i_stCurrentBeamParams := stCurBeamParams,
	i_stMachineTargetBeamParams := stMachineTargetBeamParams,
	i_stRequestedBeamParams := stReqBeamParams,
	io_fbFFHWO := fbFFO);
	
fbFFO.EvaluateOutput(q_xFastFaultOut=>q_Output);

fbAssert.AssertFalse(q_Output,
	'Limits moved beyond current and target beam, should produce a fault.');

//Beam and target eV moved back within permitted ranges, reset clears fault
stCurBeamParams.reV := 300;
	
stMachineTargetBeamParams.reV := 300;

stReqBeamParams.neVReqRange := 2#0000_1111_0011_1111;

fbFFO(i_xReset:=TRUE); //New reset request

fbPEW.i_xReset := TRUE; //New reset request

fbPEW(i_stCurrentBeamParams := stCurBeamParams, //Beam params are now within spec
	i_stMachineTargetBeamParams := stMachineTargetBeamParams,
	i_stRequestedBeamParams := stReqBeamParams,
	io_fbFFHWO := fbFFO);
	
fbFFO.EvaluateOutput(q_xFastFaultOut=>q_Output);

fbAssert.AssertTrue(q_Output,
	'Beam within limits after reset, FFO should be true');
	
//At this point, the fast fault would be cleared

//Current beam eV moved out of range
stCurBeamParams.reV := 800; //Moved out of range
	
stMachineTargetBeamParams.reV := 300; //Still within range

stReqBeamParams.neVReqRange := 2#0000_1111_0011_1111;

fbPEW(i_stCurrentBeamParams := stCurBeamParams,
	i_stMachineTargetBeamParams := stMachineTargetBeamParams,
	i_stRequestedBeamParams := stReqBeamParams,
	io_fbFFHWO := fbFFO);
	
fbFFO.EvaluateOutput(q_xFastFaultOut=>q_Output);

fbAssert.AssertFalse(q_Output,
	'Current beam moved beyond set limits, should produce a fault');

//Target beam eV moved out of range
fbFFO(i_xReset:=FALSE); //Reset released
fbFFO(i_xReset:=TRUE); //New reset request comes in at the top of a cycle, but will be overridden

stCurBeamParams.reV := 300; //Now within range
	
stMachineTargetBeamParams.reV := 800; //Moved out of range

stReqBeamParams.neVReqRange := 2#0000_1111_0011_1111;

fbPEW.i_xReset := TRUE; //Attempt to reset local FF will fail
fbPEW(i_stCurrentBeamParams := stCurBeamParams,
	i_stMachineTargetBeamParams := stMachineTargetBeamParams,
	i_stRequestedBeamParams := stReqBeamParams,
	io_fbFFHWO := fbFFO);
	
fbFFO.EvaluateOutput(q_xFastFaultOut=>q_Output);

fbAssert.AssertFalse(q_Output,
	'Target beam moved beyond set limits, should produce a fault');
END_METHOD

METHOD RunTests : TCUNIT.E_TestSuiteRunState
PEWatcherBasicFunction();

RunTests := TcUnit.E_TestSuiteRunState.FINISHED;
END_METHOD

END_FUNCTION_BLOCK

// POUs/TestComponents/FB_SafeBPCompare_Test
{attribute 'call_after_init'}
FUNCTION_BLOCK FB_SafeBPCompare_Test EXTENDS FB_TestSuite IMPLEMENTS I_RunnableTestSuite
VAR_INPUT
END_VAR
VAR_OUTPUT
END_VAR
VAR
	fbAssert : TcUnit.FB_Assert;
END_VAR

//Verify beam off is considered safe.
METHOD PRIVATE BeamOffIsSafe
VAR_INPUT
END_VAR
VAR
	stBeamOn	:	ST_BeamParams;
	stBeamOff	:	ST_BeamParams;
	
END_VAR
stBeamOn := F_SetBeamParams(
	50, //50% attenuation is more conservative than 0
	10,
	16#FFFF,
	120);

stBeamOff := F_SetBeamParams(
	0, //0% attenuation
	10,
	16#FFFF,
	0); //0 beam rate means this bps is actually safer than BeamOn

TEST('BeamOffIsSafe');
	
fbAssert.AssertTrue(
	F_SafeBPCompare(stBeamOff, stBeamOn),
	'SafeBPCompare does not think beam rate = 0 is safer than anything else.');
END_METHOD

//Verify BP comparison remains logical.
METHOD PRIVATE BPComparisonCheck
VAR_INPUT
END_VAR
VAR
	stSafer	:	ST_BeamParams;
	stNotSoSafe	:	ST_BeamParams;
END_VAR
TEST('BPComparisonCheck');


//Attenuation
stSafer := F_SetBeamParams(
	1, //
	10,
	16#FFFF,
	1);

stNotSoSafe := F_SetBeamParams(
	0, //
	10,
	16#FFFF,
	1); 
	
fbAssert.AssertTrue(
	F_SafeBPCompare(stSafer, stNotSoSafe),
	'Attenuation eval is broken (True)'); 

fbAssert.AssertFalse(
	F_SafeBPCompare(stNotSoSafe, stSafer),
	'Attenuation eval is broken (False)');
	
	
//Rate
stSafer := F_SetBeamParams(
	0,
	10,
	16#FFFF,
	1); //

stNotSoSafe := F_SetBeamParams(
	0,
	10,
	16#FFFF,
	10); //
	
fbAssert.AssertTrue(
	F_SafeBPCompare(stSafer, stNotSoSafe),
	'Rate eval is broken (True)'); 

fbAssert.AssertFalse(
	F_SafeBPCompare(stNotSoSafe, stSafer),
	'Rate eval is broken (False)');
	
//Pulse energy
stSafer := F_SetBeamParams(
	0, 
	1, //
	16#FFFF,
	1);

stNotSoSafe := F_SetBeamParams(
	0, 
	10, //
	16#FFFF,
	1); 
	
fbAssert.AssertTrue(
	F_SafeBPCompare(stSafer, stNotSoSafe),
	'Pulse energy eval is broken (True)'); 

fbAssert.AssertFalse(
	F_SafeBPCompare(stNotSoSafe, stSafer),
	'Pulse energy eval is broken (False)');	
	
//Photon energy
//More extensive tests elsewhere
stSafer := F_SetBeamParams(
	0, 
	1, 
	2#0000_0000_0000_0110, //200-400eV
	1);
	
stSafer.reV := 300; //

stNotSoSafe := F_SetBeamParams(
	0, 
	1, 
	2#0000_0000_0000_0110, //200-400ev
	1);
	
stNotSoSafe.reV := 401;
	
fbAssert.AssertTrue(
	F_SafeBPCompare(stSafer, stNotSoSafe),
	'Photon energy eval is broken (True)'); 

fbAssert.AssertFalse(
	F_SafeBPCompare(stNotSoSafe, stSafer),
	'Photon energy eval is broken (False)');
END_METHOD

METHOD FB_init : BOOL
VAR_INPUT
	bInitRetains : BOOL; // if TRUE, the retain variables are initialized (warm start / cold start)
	bInCopyCode : BOOL;  // if TRUE, the instance afterwards gets moved into the copy code (online change)
END_VAR
SUPER^.RegisterTestSuite(THIS^);
END_METHOD

METHOD RunTests : TCUNIT.E_TestSuiteRunState
BeamOffIsSafe();
BPComparisonCheck();

RunTests := TcUnit.E_TestSuiteRunState.FINISHED;
END_METHOD

END_FUNCTION_BLOCK

// POUs/TestComponents/FB_SolidAttenuator
FUNCTION_BLOCK FB_SolidAttenuator
VAR_INPUT
	i_rRequestedAttenuation	:	REAL;
END_VAR
VAR_OUTPUT
	q_xFault	:	BOOL;
	q_rCurrentAttenuation	:	REAL;
END_VAR
VAR_IN_OUT
	Arbiter	:	FB_Arbiter; //Higher level arbiter from which upstream attenuation can be requested
END_VAR
VAR
	stAttenuator	:	ST_BinarySolidAttenuator;
	nSearchStart: INT;
	nArrayLength: INT;
	axNewBladeStates	:	ARRAY [0..9]	OF	BOOL;
	nTryIndex: INT;
	rCurrentAccumulatedAttenuation: REAL;
	rTryFilter: REAL;
	rTryAttenuation: REAL;
	rRequestedAttenuation: REAL;
END_VAR



//

//Assuming the blades are ordered thickest to thinnest 
REPEAT
	rTryAttenuation := rCurrentAccumulatedAttenuation + stAttenuator.axBlades[nTryIndex].rThickness;
	IF rRequestedAttenuation >= rTryAttenuation THEN
		rCurrentAccumulatedAttenuation := rTryAttenuation;
		axNewBladeStates[nTryIndex] := TRUE;
	ELSE
		axNewBladeStates[nTryIndex] := FALSE;
	END_IF
UNTIL
	nTryIndex >= nArrayLength
END_REPEAT

END_FUNCTION_BLOCK

// POUs/Fast_Faults
PROGRAM Fast_Faults
VAR
END_VAR

g_FastFaultOutput1();

END_PROGRAM

// POUs/Fast_Faults_Evaluate
PROGRAM Fast_Faults_Evaluate
VAR
END_VAR

g_FastFaultOutput1.EvaluateOutput();

END_PROGRAM

// POUs/MachineSimulation
PROGRAM MachineSimulation
VAR
	fbMachine	:	FB_MachineSimulator;
END_VAR

//Machine simulator
fbMachine(
	i_stAssertedParams := g_fbArbiter.q_stBeamParams,
	q_stMachineParams => PMPS_GVL_BeamParams.stCurrentBeamParameters,
	i_xFault	:= NOT GVL.g_FastFaultOutput1.q_xFastFaultOut
	);

END_PROGRAM

// POUs/MAIN
PROGRAM MAIN
VAR
	fbDev1	:	FB_ExampleDeviceSM_All;
	fbDev2	:	FB_ExampleDeviceSM_All;
	
	rtInit	:	R_TRIG;
	Initialize	:	BOOL := TRUE;
	
	DemoMode: BOOL;
END_VAR

//Sub-system Device PLC

IF DemoMode	THEN

//Fast Faults must run first
Fast_Faults();

IF Initialize THEN
	fbDev1(cBase := 10,
		fbFastFaultOutput := g_FastFaultOutput1,
		fbArbiter := g_fbArbiter);
	fbDev2(cBase := 1000,
		fbFastFaultOutput := g_FastFaultOutput1,
		fbArbiter := g_fbArbiter);
	g_fbArbiter.A_Init();
	Initialize := FALSE;
END_IF

//Example devices
fbDev1(fbFastFaultOutput := g_FastFaultOutput1,
		fbArbiter := g_fbArbiter);
fbDev2(fbFastFaultOutput := g_FastFaultOutput1,
		fbArbiter := g_fbArbiter);


PMPS_Arbiter();

Fast_Faults_Evaluate();

MachineSimulation();

ELSE
	TestSetups();
END_IF

ACTION Initialize:

END_ACTION

END_PROGRAM

// POUs/PMPS_Arbiter
PROGRAM PMPS_Arbiter
VAR
	
	
	
	
	fbPhotonEnergyWatcher	:	FB_PhotonEnergyWatcher;
	
	fbMPSInterface	:	FB_BeamClassOutputs;
	{attribute 'pmps_interface' := 'TIID^Device 2 (EtherCAT)^Term 6 (EK1100)^Term 2 (EL6692)^IO Outputs^'}
	ExchangeBeamParams	:	FB_BeamParamEx;
END_VAR


//Execute arbiter
g_fbArbiter.q_stBeamParams:= g_fbArbiter.GetArbitratedBP();

//fbMPSInterface();

fbPhotonEnergyWatcher(i_stCurrentBeamParams	:= PMPS_GVL_BeamParams.stCurrentBeamParameters,
					i_stRequestedBeamParams := g_fbArbiter.q_stBeamParams,
					io_fbFFHWO:= GVL.g_FastFaultOutput1);

ExchangeBeamParams();

END_PROGRAM

// POUs/TestSetups
//Test setups (fixtures), for PMPS components
PROGRAM TestSetups
VAR
	fbBPTMTest	:	FB_BPTM_Test;
	fbSafeBPCompareTest	:	FB_SafeBPCompare_Test;
	fbevWithinSpecTest	:	FB_evWithinSpec_Test;
	fbPEWTest	:	FB_PhotonEnergyWatcher_Test;
	fbFFTest	:	FB_FastFault_Test;
	fbArbiterTest	:	FB_Arbiter_Test;
END_VAR

TcUnit.RUN();

END_PROGRAM

// VISUs/ArbiterStats
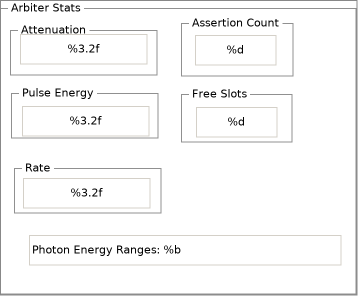
VISUALIZATION ArbiterStats  // 358x296
VAR_IN_OUT
	fbArbiter	:	FB_Arbiter;
END_VAR
    GroupBox (0,0 356x294), "Arbiter Stats"
        GroupBox (10,22 147x53), "Attenuation"
            Textfield (10,12 127x30), "%3.2f", text variable: fbArbiter.q_stBeamParams.fAtt
        GroupBox (11,85 147x53), "Pulse Energy"
            Textfield (11,21 127x30), "%3.2f", text variable: fbArbiter.q_stBeamParams.fPP_mJ
        GroupBox (14,160 147x53), "Rate"
            Textfield (9,18 127x30), "%3.2f", text variable: fbArbiter.stOutputBP.nRate
        GroupBox (181,15 112x61), "Assertion Count"
            Textfield (14,20 81x30), "%d", text variable: fbArbiter.fbBPAssertionPool.hTable.nCount
        GroupBox (181,86 111x56), "Free Slots"
            Textfield (15,21 81x30), "%d", text variable: fbArbiter.fbBPAssertionPool.hTable.nFree
        Textfield (29,235 312x30), "Photon Energy Ranges: %b", text variable: fbArbiter.q_stBeamParams.neVReqRange
END_VISUALIZATION

// VISUs/FastFaultGUI
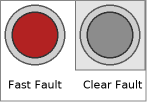
VISUALIZATION FastFaultGUI  // 147x102
VAR_IN_OUT
	FastFault	:	FB_HardwareFFOutput;
END_VAR
    Lamp1 (0,0 70x70), variable: NOT FastFault.q_xFastFaultOut, style: Lamp-Lamp1-Red
    Label (5,70 59x30), "Fast Fault"
    PushSwitch (75,0 70x70), variable: FastFault.i_xReset, behaviour: TAP, style: Switch-PushSwitch-Gray
    Label (80,70 59x30), "Clear Fault"
END_VISUALIZATION

// VISUs/ImagerGUI
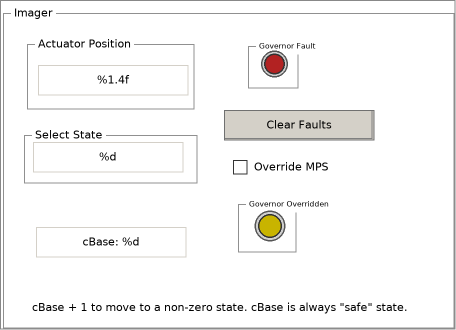
VISUALIZATION ImagerGUI  // 456x330
VAR_IN_OUT
	fbDevice	:	FB_ExampleDeviceSM_All;
END_VAR
    GroupBox (3,5 451x323), "Imager"
        Button (221,105 150x30), "Clear Faults"
            tap fbDevice.stDevice.xClearFaults
        Checkbox (228,147 150x30), "Override MPS", variable: fbDevice.stDevice.xOverrideMPSLimits
        GroupBox (245,33 50x50), "Governor Fault"
            Lamp1 (11,10 31x32), variable: fbDevice.stDevice.xGovernorFault, style: Lamp-Lamp1-Red
        GroupBox (235,191 58x56), "Governor Overridden"
            Lamp1 (14,10 36x40), variable: fbDevice.stDevice.xGovernorOverridden, style: Lamp-Lamp1-Yellow
        GroupBox (24,31 167x73), "Actuator Position"
            Textfield (11,29 150x30), "%1.4f", text variable: fbDevice.stDevice.stAxis.NcToPlc.ActPos
        GroupBox (21,122 173x56), "Select State"
            Textfield (9,15 150x30), "%d", tooltip "cBase + 1 to move to a non-zero state. cBase is always "safe" state.", text variable: fbDevice.stDevice.nRequestedState
                OnMouseDown: write the text variable via Default
        Label (33,293 368x19), "cBase + 1 to move to a non-zero state. cBase is always "safe" state."
        Textfield (33,222 150x30), "cBase: %d", tooltip "cBase + 1 to move to a non-zero state. cBase is always "safe" state.", text variable: fbDevice.cBase
            OnMouseDown: write the text variable via Default
END_VISUALIZATION

// VISUs/PhotonEnergyWatcher
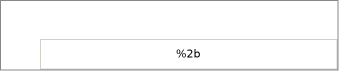
VISUALIZATION PhotonEnergyWatcher  // 339x71
VAR_IN_OUT
	Watcher	:	FB_PhotonEnergyWatcher;
END_VAR
    Textfield (40,39 297x30), "%2b", text variable: Watcher.i_stCurrentBeamParams.neVReqRange
END_VISUALIZATION

// VISUs/Visualization
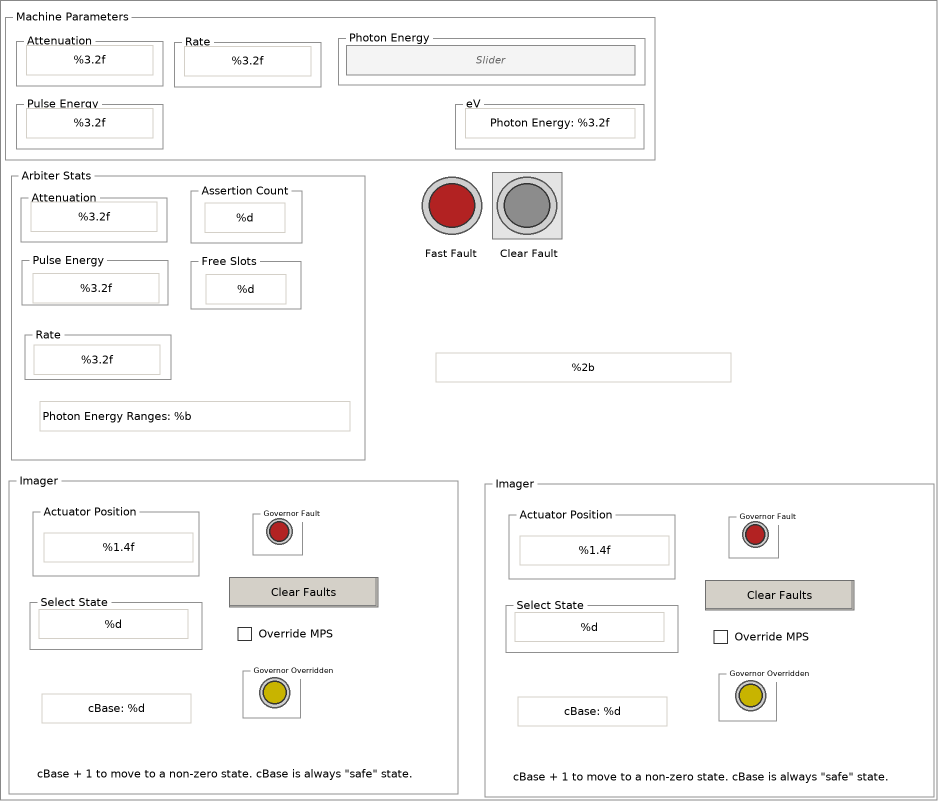
VISUALIZATION Visualization  // 938x801
    GroupBox (5,9 650x151), "Machine Parameters"
        GroupBox (11,24 147x53), "Attenuation"
            Textfield (10,12 127x30), "%3.2f", text variable: PMPS_GVL_BeamParams.stCurrentBeamParameters.fAtt
        GroupBox (11,87 147x53), "Pulse Energy"
            Textfield (10,12 127x30), "%3.2f", text variable: PMPS_GVL_BeamParams.stCurrentBeamParameters.fPP_mJ
        GroupBox (169,25 147x53), "Rate"
            Textfield (10,12 127x30), "%3.2f", text variable: PMPS_GVL_BeamParams.stCurrentBeamParameters.nRate
        GroupBox (333,21 307x55), "Photon Energy"
            Slider (8,15 289x30), variable: MachineSimulation.fbMachine.i_reV, scale 0..1600
        GroupBox (450,87 189x53), "eV"
            Textfield (10,12 170x30), "Photon Energy: %3.2f", text variable: PMPS_GVL_BeamParams.stCurrentBeamParameters.reV
    Frame (6,468 454x328)
        shows ImagerGUI(fbDevice := MAIN.fbDev1)
    Frame (482,471 454x328)
        shows ImagerGUI(fbDevice := MAIN.fbDev2)
    Frame (417,172 147x98)
        shows FastFaultGUI(FastFault := GVL.g_FastFaultOutput1)
    Frame (11,168 356x294)
        shows ArbiterStats(fbArbiter := GVL.g_fbArbiter)
    Frame (396,315 337x69)
        shows PhotonEnergyWatcher(Watcher := PMPS_Arbiter.fbPhotonEnergyWatcher)
END_VISUALIZATION
